// TIA Portal project "olbu" (V15)

(* hardware
DEVICE "S71500/ET200MP station_1"  S7-1500 station
   slot 0: "Rail_0"  Rack  6ES7 590-1***0-0AA0
   slot 1: "PLC_1"  CPU 1517F-3 PN/DP  6ES7 517-3FP00-0AB0  V2.5
      slot 3: "CPU display_1"  6ES7591-1BA00-0AA0
DEVICE "ET 200SP station_1"  ET 200SP-Station
   slot 0: "Rack_0"  Rack  6ES5 710-8MAx1
   slot 0: "volvo1606et200sp"  IM 155-6 PN ST  6ES7 155-6AU01-0BN0  V4.1
   slot 1: "DQ 8x24VDC/0.5A ST_1"  DQ 8x24VDC/0.5A ST  6ES7 132-6BF01-0BA0  V0.0
      slot 1: "DQ 8x24VDC/0.5A ST_1"  DQ 8x24VDC/0.5A ST
   slot 2: "DQ 8x24VDC/0.5A ST_2"  DQ 8x24VDC/0.5A ST  6ES7 132-6BF01-0BA0  V0.0
      slot 1: "DQ 8x24VDC/0.5A ST_2"  DQ 8x24VDC/0.5A ST
   slot 3: "DQ 8x24VDC/0.5A ST_3"  DQ 8x24VDC/0.5A ST  6ES7 132-6BF01-0BA0  V0.0
      slot 1: "DQ 8x24VDC/0.5A ST_3"  DQ 8x24VDC/0.5A ST
   slot 4: "Server module_1"  Server module  6ES7 193-6PA00-0AA0  V1.1
      slot 1: "Server module_1"  Server module
   slot 127: "BA 2xRJ45"  BA 2xRJ45  6ES7 193-6AR00-0AA0  V0.0
      slot 1: "Port_1"  6ES7 193-6AR00-0AA0  V0.0
      slot 2: "Port_2"  6ES7 193-6AR00-0AA0  V0.0
DEVICE "ET 200SP station_2"  ET 200SP-Station
   slot 0: "Rack_0"  Rack  6ES5 710-8MAx1
   slot 0: "volvo1607et200sp"  IM 155-6 PN ST  6ES7 155-6AU01-0BN0  V4.1
   slot 1: "DQ 8x24VDC/0.5A ST_1"  DQ 8x24VDC/0.5A ST  6ES7 132-6BF01-0BA0  V0.0
      slot 1: "DQ 8x24VDC/0.5A ST_1"  DQ 8x24VDC/0.5A ST
   slot 2: "DQ 8x24VDC/0.5A ST_2"  DQ 8x24VDC/0.5A ST  6ES7 132-6BF01-0BA0  V0.0
      slot 1: "DQ 8x24VDC/0.5A ST_2"  DQ 8x24VDC/0.5A ST
   slot 3: "DQ 8x24VDC/0.5A ST_3"  DQ 8x24VDC/0.5A ST  6ES7 132-6BF01-0BA0  V0.0
      slot 1: "DQ 8x24VDC/0.5A ST_3"  DQ 8x24VDC/0.5A ST
   slot 4: "Server module_1"  Server module  6ES7 193-6PA00-0AA0  V1.1
      slot 1: "Server module_1"  Server module
   slot 127: "BA 2xRJ45"  BA 2xRJ45  6ES7 193-6AR00-0AA0  V0.0
      slot 1: "Port_1"  6ES7 193-6AR00-0AA0  V0.0
      slot 2: "Port_2"  6ES7 193-6AR00-0AA0  V0.0
DEVICE "ET 200SP station_3"  ET 200SP-Station
   slot 0: "Rack_0"  Rack  6ES5 710-8MAx1
   slot 0: "volvo1608et200sp"  IM 155-6 PN ST  6ES7 155-6AU01-0BN0  V4.1
   slot 1: "DQ 8x24VDC/0.5A ST_1"  DQ 8x24VDC/0.5A ST  6ES7 132-6BF01-0BA0  V0.0
      slot 1: "DQ 8x24VDC/0.5A ST_1"  DQ 8x24VDC/0.5A ST
   slot 2: "DQ 8x24VDC/0.5A ST_2"  DQ 8x24VDC/0.5A ST  6ES7 132-6BF01-0BA0  V0.0
      slot 1: "DQ 8x24VDC/0.5A ST_2"  DQ 8x24VDC/0.5A ST
   slot 3: "DQ 8x24VDC/0.5A ST_3"  DQ 8x24VDC/0.5A ST  6ES7 132-6BF01-0BA0  V0.0
      slot 1: "DQ 8x24VDC/0.5A ST_3"  DQ 8x24VDC/0.5A ST
   slot 4: "Server module_1"  Server module  6ES7 193-6PA00-0AA0  V1.1
      slot 1: "Server module_1"  Server module
   slot 127: "BA 2xRJ45"  BA 2xRJ45  6ES7 193-6AR00-0AA0  V0.0
      slot 1: "Port_1"  6ES7 193-6AR00-0AA0  V0.0
      slot 2: "Port_2"  6ES7 193-6AR00-0AA0  V0.0
DEVICE "KP8_1"  SIMATIC Key Panel
   slot 0: "Rack"  Rail  V1.0
   slot 0: "volvo1608kp8"  KP8  6AV3 688-3AY36-0AX0  R01.00.00
DEVICE "KP8_2"  SIMATIC Key Panel
   slot 0: "Rack"  Rail  V1.0
   slot 0: "volvo1607kp8"  KP8  6AV3 688-3AY36-0AX0  R01.00.00
DEVICE "KP8_3"  SIMATIC Key Panel
   slot 0: "Rack"  Rail  V1.0
   slot 0: "volvo1606kp8"  KP8  6AV3 688-3AY36-0AX0  R01.00.00
DEVICE "KP8_4"  SIMATIC Key Panel
   slot 0: "Rack"  Rail  V1.0
   slot 0: "volvo1609kp8"  KP8  6AV3 688-3AY36-0AX0  R01.00.00
DEVICE "ET 200SP station_4"  ET 200SP-Station
   slot 0: "Rack_0"  Rack  6ES5 710-8MAx1
   slot 0: "volvo1609et200sp"  IM 155-6 PN ST  6ES7 155-6AU01-0BN0  V4.1
   slot 1: "DQ 8x24VDC/0.5A ST_1"  DQ 8x24VDC/0.5A ST  6ES7 132-6BF01-0BA0  V0.0
      slot 1: "DQ 8x24VDC/0.5A ST_1"  DQ 8x24VDC/0.5A ST
   slot 2: "DQ 8x24VDC/0.5A ST_2"  DQ 8x24VDC/0.5A ST  6ES7 132-6BF01-0BA0  V0.0
      slot 1: "DQ 8x24VDC/0.5A ST_2"  DQ 8x24VDC/0.5A ST
   slot 3: "DQ 8x24VDC/0.5A ST_3"  DQ 8x24VDC/0.5A ST  6ES7 132-6BF01-0BA0  V0.0
      slot 1: "DQ 8x24VDC/0.5A ST_3"  DQ 8x24VDC/0.5A ST
   slot 4: "Server module_1"  Server module  6ES7 193-6PA00-0AA0  V1.1
      slot 1: "Server module_1"  Server module
   slot 127: "BA 2xRJ45"  BA 2xRJ45  6ES7 193-6AR00-0AA0  V0.0
      slot 1: "Port_1"  6ES7 193-6AR00-0AA0  V0.0
      slot 2: "Port_2"  6ES7 193-6AR00-0AA0  V0.0
DEVICE "ET 200SP station_5"  ET 200SP-Station
   slot 0: "Rack_0"  Rack  6ES5 710-8MAx1
   slot 0: "volvo1610et200sp"  IM 155-6 PN ST  6ES7 155-6AU01-0BN0  V4.1
   slot 1: "DQ 8x24VDC/0.5A ST_1"  DQ 8x24VDC/0.5A ST  6ES7 132-6BF01-0BA0  V0.0
      slot 1: "DQ 8x24VDC/0.5A ST_1"  DQ 8x24VDC/0.5A ST
   slot 2: "DQ 8x24VDC/0.5A ST_2"  DQ 8x24VDC/0.5A ST  6ES7 132-6BF01-0BA0  V0.0
      slot 1: "DQ 8x24VDC/0.5A ST_2"  DQ 8x24VDC/0.5A ST
   slot 3: "DQ 8x24VDC/0.5A ST_3"  DQ 8x24VDC/0.5A ST  6ES7 132-6BF01-0BA0  V0.0
      slot 1: "DQ 8x24VDC/0.5A ST_3"  DQ 8x24VDC/0.5A ST
   slot 4: "Server module_1"  Server module  6ES7 193-6PA00-0AA0  V1.1
      slot 1: "Server module_1"  Server module
   slot 127: "BA 2xRJ45"  BA 2xRJ45  6ES7 193-6AR00-0AA0  V0.0
      slot 1: "Port_1"  6ES7 193-6AR00-0AA0  V0.0
      slot 2: "Port_2"  6ES7 193-6AR00-0AA0  V0.0
DEVICE "KP8_5"  SIMATIC Key Panel
   slot 0: "Rack"  Rail  V1.0
   slot 0: "volvo1610kp8"  KP8  6AV3 688-3AY36-0AX0  R01.00.00
DEVICE "ET 200SP station_6"  ET 200SP-Station
   slot 0: "Rack_0"  Rack  6ES5 710-8MAx1
   slot 0: "volvo1611et200sp"  IM 155-6 PN ST  6ES7 155-6AU01-0BN0  V4.1
   slot 1: "DQ 8x24VDC/0.5A ST_1"  DQ 8x24VDC/0.5A ST  6ES7 132-6BF01-0BA0  V0.0
      slot 1: "DQ 8x24VDC/0.5A ST_1"  DQ 8x24VDC/0.5A ST
   slot 2: "DQ 8x24VDC/0.5A ST_2"  DQ 8x24VDC/0.5A ST  6ES7 132-6BF01-0BA0  V0.0
      slot 1: "DQ 8x24VDC/0.5A ST_2"  DQ 8x24VDC/0.5A ST
   slot 3: "DQ 8x24VDC/0.5A ST_3"  DQ 8x24VDC/0.5A ST  6ES7 132-6BF01-0BA0  V0.0
      slot 1: "DQ 8x24VDC/0.5A ST_3"  DQ 8x24VDC/0.5A ST
   slot 4: "Server module_1"  Server module  6ES7 193-6PA00-0AA0  V1.1
      slot 1: "Server module_1"  Server module
   slot 127: "BA 2xRJ45"  BA 2xRJ45  6ES7 193-6AR00-0AA0  V0.0
      slot 1: "Port_1"  6ES7 193-6AR00-0AA0  V0.0
      slot 2: "Port_2"  6ES7 193-6AR00-0AA0  V0.0
DEVICE "KP8_6"  SIMATIC Key Panel
   slot 0: "Rack"  Rail  V1.0
   slot 0: "volvo1611kp8"  KP8  6AV3 688-3AY36-0AX0  R01.00.00
DEVICE "KP8_7"  SIMATIC Key Panel
   slot 0: "Rack"  Rail  V1.0
   slot 0: "volvo1601kp8"  KP8  6AV3 688-3AY36-0AX0  R01.00.00
DEVICE "ET 200SP station_7"  ET 200SP-Station
   slot 0: "Rack_0"  Rack  6ES5 710-8MAx1
   slot 0: "volvo1601et200sp"  IM 155-6 PN ST  6ES7 155-6AU01-0BN0  V4.1
   slot 1: "DQ 8x24VDC/0.5A ST_1"  DQ 8x24VDC/0.5A ST  6ES7 132-6BF01-0BA0  V0.0
      slot 1: "DQ 8x24VDC/0.5A ST_1"  DQ 8x24VDC/0.5A ST
   slot 2: "DQ 8x24VDC/0.5A ST_2"  DQ 8x24VDC/0.5A ST  6ES7 132-6BF01-0BA0  V0.0
      slot 1: "DQ 8x24VDC/0.5A ST_2"  DQ 8x24VDC/0.5A ST
   slot 3: "DQ 8x24VDC/0.5A ST_3"  DQ 8x24VDC/0.5A ST  6ES7 132-6BF01-0BA0  V0.0
      slot 1: "DQ 8x24VDC/0.5A ST_3"  DQ 8x24VDC/0.5A ST
   slot 4: "Server module_1"  Server module  6ES7 193-6PA00-0AA0  V1.1
      slot 1: "Server module_1"  Server module
   slot 127: "BA 2xRJ45"  BA 2xRJ45  6ES7 193-6AR00-0AA0  V0.0
      slot 1: "Port_1"  6ES7 193-6AR00-0AA0  V0.0
      slot 2: "Port_2"  6ES7 193-6AR00-0AA0  V0.0
DEVICE "KP8_8"  SIMATIC Key Panel
   slot 0: "Rack"  Rail  V1.0
   slot 0: "volvo1602kp8"  KP8  6AV3 688-3AY36-0AX0  R01.00.00
DEVICE "ET 200SP station_8"  ET 200SP-Station
   slot 0: "Rack_0"  Rack  6ES5 710-8MAx1
   slot 0: "volvo1602et200sp"  IM 155-6 PN ST  6ES7 155-6AU01-0BN0  V4.1
   slot 1: "DQ 8x24VDC/0.5A ST_1"  DQ 8x24VDC/0.5A ST  6ES7 132-6BF01-0BA0  V0.0
      slot 1: "DQ 8x24VDC/0.5A ST_1"  DQ 8x24VDC/0.5A ST
   slot 2: "DQ 8x24VDC/0.5A ST_2"  DQ 8x24VDC/0.5A ST  6ES7 132-6BF01-0BA0  V0.0
      slot 1: "DQ 8x24VDC/0.5A ST_2"  DQ 8x24VDC/0.5A ST
   slot 3: "DQ 8x24VDC/0.5A ST_3"  DQ 8x24VDC/0.5A ST  6ES7 132-6BF01-0BA0  V0.0
      slot 1: "DQ 8x24VDC/0.5A ST_3"  DQ 8x24VDC/0.5A ST
   slot 4: "Server module_1"  Server module  6ES7 193-6PA00-0AA0  V1.1
      slot 1: "Server module_1"  Server module
   slot 127: "BA 2xRJ45"  BA 2xRJ45  6ES7 193-6AR00-0AA0  V0.0
      slot 1: "Port_1"  6ES7 193-6AR00-0AA0  V0.0
      slot 2: "Port_2"  6ES7 193-6AR00-0AA0  V0.0
DEVICE "KP8_9"  SIMATIC Key Panel
   slot 0: "Rack"  Rail  V1.0
   slot 0: "volvo1603kp8"  KP8  6AV3 688-3AY36-0AX0  R01.00.00
DEVICE "ET 200SP station_9"  ET 200SP-Station
   slot 0: "Rack_0"  Rack  6ES5 710-8MAx1
   slot 0: "volvo1603et200sp"  IM 155-6 PN ST  6ES7 155-6AU01-0BN0  V4.1
   slot 1: "DQ 8x24VDC/0.5A ST_1"  DQ 8x24VDC/0.5A ST  6ES7 132-6BF01-0BA0  V0.0
      slot 1: "DQ 8x24VDC/0.5A ST_1"  DQ 8x24VDC/0.5A ST
   slot 2: "DQ 8x24VDC/0.5A ST_2"  DQ 8x24VDC/0.5A ST  6ES7 132-6BF01-0BA0  V0.0
      slot 1: "DQ 8x24VDC/0.5A ST_2"  DQ 8x24VDC/0.5A ST
   slot 3: "DQ 8x24VDC/0.5A ST_3"  DQ 8x24VDC/0.5A ST  6ES7 132-6BF01-0BA0  V0.0
      slot 1: "DQ 8x24VDC/0.5A ST_3"  DQ 8x24VDC/0.5A ST
   slot 4: "Server module_1"  Server module  6ES7 193-6PA00-0AA0  V1.1
      slot 1: "Server module_1"  Server module
   slot 127: "BA 2xRJ45"  BA 2xRJ45  6ES7 193-6AR00-0AA0  V0.0
      slot 1: "Port_1"  6ES7 193-6AR00-0AA0  V0.0
      slot 2: "Port_2"  6ES7 193-6AR00-0AA0  V0.0
DEVICE "KP8_10"  SIMATIC Key Panel
   slot 0: "Rack"  Rail  V1.0
   slot 0: "volvo1604kp8"  KP8  6AV3 688-3AY36-0AX0  R01.00.00
DEVICE "ET 200SP station_10"  ET 200SP-Station
   slot 0: "Rack_0"  Rack  6ES5 710-8MAx1
   slot 0: "volvo1604et200sp"  IM 155-6 PN ST  6ES7 155-6AU01-0BN0  V4.1
   slot 1: "DQ 8x24VDC/0.5A ST_1"  DQ 8x24VDC/0.5A ST  6ES7 132-6BF01-0BA0  V0.0
      slot 1: "DQ 8x24VDC/0.5A ST_1"  DQ 8x24VDC/0.5A ST
   slot 2: "DQ 8x24VDC/0.5A ST_2"  DQ 8x24VDC/0.5A ST  6ES7 132-6BF01-0BA0  V0.0
      slot 1: "DQ 8x24VDC/0.5A ST_2"  DQ 8x24VDC/0.5A ST
   slot 3: "DQ 8x24VDC/0.5A ST_3"  DQ 8x24VDC/0.5A ST  6ES7 132-6BF01-0BA0  V0.0
      slot 1: "DQ 8x24VDC/0.5A ST_3"  DQ 8x24VDC/0.5A ST
   slot 4: "Server module_1"  Server module  6ES7 193-6PA00-0AA0  V1.1
      slot 1: "Server module_1"  Server module
   slot 127: "BA 2xRJ45"  BA 2xRJ45  6ES7 193-6AR00-0AA0  V0.0
      slot 1: "Port_1"  6ES7 193-6AR00-0AA0  V0.0
      slot 2: "Port_2"  6ES7 193-6AR00-0AA0  V0.0
DEVICE "KP8_11"  SIMATIC Key Panel
   slot 0: "Rack"  Rail  V1.0
   slot 0: "volvo1605kp8"  KP8  6AV3 688-3AY36-0AX0  R01.00.00
DEVICE "ET 200SP station_11"  ET 200SP-Station
   slot 0: "Rack_0"  Rack  6ES5 710-8MAx1
   slot 0: "volvo1605et200sp"  IM 155-6 PN ST  6ES7 155-6AU01-0BN0  V4.1
   slot 1: "DQ 8x24VDC/0.5A ST_1"  DQ 8x24VDC/0.5A ST  6ES7 132-6BF01-0BA0  V0.0
      slot 1: "DQ 8x24VDC/0.5A ST_1"  DQ 8x24VDC/0.5A ST
   slot 2: "DQ 8x24VDC/0.5A ST_2"  DQ 8x24VDC/0.5A ST  6ES7 132-6BF01-0BA0  V0.0
      slot 1: "DQ 8x24VDC/0.5A ST_2"  DQ 8x24VDC/0.5A ST
   slot 3: "DQ 8x24VDC/0.5A ST_3"  DQ 8x24VDC/0.5A ST  6ES7 132-6BF01-0BA0  V0.0
      slot 1: "DQ 8x24VDC/0.5A ST_3"  DQ 8x24VDC/0.5A ST
   slot 4: "Server module_1"  Server module  6ES7 193-6PA00-0AA0  V1.1
      slot 1: "Server module_1"  Server module
   slot 127: "BA 2xRJ45"  BA 2xRJ45  6ES7 193-6AR00-0AA0  V0.0
      slot 1: "Port_1"  6ES7 193-6AR00-0AA0  V0.0
      slot 2: "Port_2"  6ES7 193-6AR00-0AA0  V0.0
DEVICE "KP8_12"  SIMATIC Key Panel
   slot 0: "Rack"  Rail  V1.0
   slot 0: "chm02kp8"  KP8  6AV3 688-3AY36-0AX0  R01.00.00
DEVICE "ET 200SP station_12"  ET 200SP-Station
   slot 0: "Rack_0"  Rack  6ES5 710-8MAx1
   slot 0: "chm02et200sp"  IM 155-6 PN ST  6ES7 155-6AU01-0BN0  V4.1
   slot 1: "DQ 8x24VDC/0.5A ST_1"  DQ 8x24VDC/0.5A ST  6ES7 132-6BF01-0BA0  V0.0
      slot 1: "DQ 8x24VDC/0.5A ST_1"  DQ 8x24VDC/0.5A ST
   slot 2: "DQ 8x24VDC/0.5A ST_2"  DQ 8x24VDC/0.5A ST  6ES7 132-6BF01-0BA0  V0.0
      slot 1: "DQ 8x24VDC/0.5A ST_2"  DQ 8x24VDC/0.5A ST
   slot 3: "DQ 8x24VDC/0.5A ST_3"  DQ 8x24VDC/0.5A ST  6ES7 132-6BF01-0BA0  V0.0
      slot 1: "DQ 8x24VDC/0.5A ST_3"  DQ 8x24VDC/0.5A ST
   slot 4: "Server module_1"  Server module  6ES7 193-6PA00-0AA0  V1.1
      slot 1: "Server module_1"  Server module
   slot 127: "BA 2xRJ45"  BA 2xRJ45  6ES7 193-6AR00-0AA0  V0.0
      slot 1: "Port_1"  6ES7 193-6AR00-0AA0  V0.0
      slot 2: "Port_2"  6ES7 193-6AR00-0AA0  V0.0
DEVICE "KP8_13"  SIMATIC Key Panel
   slot 0: "Rack"  Rail  V1.0
   slot 0: "chm03kp8"  KP8  6AV3 688-3AY36-0AX0  R01.00.00
DEVICE "ET 200SP station_13"  ET 200SP-Station
   slot 0: "Rack_0"  Rack  6ES5 710-8MAx1
   slot 0: "chm03et200sp"  IM 155-6 PN ST  6ES7 155-6AU01-0BN0  V4.1
   slot 1: "DQ 8x24VDC/0.5A ST_1"  DQ 8x24VDC/0.5A ST  6ES7 132-6BF01-0BA0  V0.0
      slot 1: "DQ 8x24VDC/0.5A ST_1"  DQ 8x24VDC/0.5A ST
   slot 2: "DQ 8x24VDC/0.5A ST_2"  DQ 8x24VDC/0.5A ST  6ES7 132-6BF01-0BA0  V0.0
      slot 1: "DQ 8x24VDC/0.5A ST_2"  DQ 8x24VDC/0.5A ST
   slot 3: "DQ 8x24VDC/0.5A ST_3"  DQ 8x24VDC/0.5A ST  6ES7 132-6BF01-0BA0  V0.0
      slot 1: "DQ 8x24VDC/0.5A ST_3"  DQ 8x24VDC/0.5A ST
   slot 4: "Server module_1"  Server module  6ES7 193-6PA00-0AA0  V1.1
      slot 1: "Server module_1"  Server module
   slot 127: "BA 2xRJ45"  BA 2xRJ45  6ES7 193-6AR00-0AA0  V0.0
      slot 1: "Port_1"  6ES7 193-6AR00-0AA0  V0.0
      slot 2: "Port_2"  6ES7 193-6AR00-0AA0  V0.0
DEVICE "KP8_14"  SIMATIC Key Panel
   slot 0: "Rack"  Rail  V1.0
   slot 0: "chm04kp8"  KP8  6AV3 688-3AY36-0AX0  R01.00.00
DEVICE "ET 200SP station_14"  ET 200SP-Station
   slot 0: "Rack_0"  Rack  6ES5 710-8MAx1
   slot 0: "chm04et200sp"  IM 155-6 PN ST  6ES7 155-6AU01-0BN0  V4.1
   slot 1: "DQ 8x24VDC/0.5A ST_1"  DQ 8x24VDC/0.5A ST  6ES7 132-6BF01-0BA0  V0.0
      slot 1: "DQ 8x24VDC/0.5A ST_1"  DQ 8x24VDC/0.5A ST
   slot 2: "DQ 8x24VDC/0.5A ST_2"  DQ 8x24VDC/0.5A ST  6ES7 132-6BF01-0BA0  V0.0
      slot 1: "DQ 8x24VDC/0.5A ST_2"  DQ 8x24VDC/0.5A ST
   slot 3: "DQ 8x24VDC/0.5A ST_3"  DQ 8x24VDC/0.5A ST  6ES7 132-6BF01-0BA0  V0.0
      slot 1: "DQ 8x24VDC/0.5A ST_3"  DQ 8x24VDC/0.5A ST
   slot 4: "Server module_1"  Server module  6ES7 193-6PA00-0AA0  V1.1
      slot 1: "Server module_1"  Server module
   slot 127: "BA 2xRJ45"  BA 2xRJ45  6ES7 193-6AR00-0AA0  V0.0
      slot 1: "Port_1"  6ES7 193-6AR00-0AA0  V0.0
      slot 2: "Port_2"  6ES7 193-6AR00-0AA0  V0.0
DEVICE "KP8_15"  SIMATIC Key Panel
   slot 0: "Rack"  Rail  V1.0
   slot 0: "chm05kp8"  KP8  6AV3 688-3AY36-0AX0  R01.00.00
DEVICE "ET 200SP station_15"  ET 200SP-Station
   slot 0: "Rack_0"  Rack  6ES5 710-8MAx1
   slot 0: "chm05et200sp"  IM 155-6 PN ST  6ES7 155-6AU01-0BN0  V4.1
   slot 1: "DQ 8x24VDC/0.5A ST_1"  DQ 8x24VDC/0.5A ST  6ES7 132-6BF01-0BA0  V0.0
      slot 1: "DQ 8x24VDC/0.5A ST_1"  DQ 8x24VDC/0.5A ST
   slot 2: "DQ 8x24VDC/0.5A ST_2"  DQ 8x24VDC/0.5A ST  6ES7 132-6BF01-0BA0  V0.0
      slot 1: "DQ 8x24VDC/0.5A ST_2"  DQ 8x24VDC/0.5A ST
   slot 3: "DQ 8x24VDC/0.5A ST_3"  DQ 8x24VDC/0.5A ST  6ES7 132-6BF01-0BA0  V0.0
      slot 1: "DQ 8x24VDC/0.5A ST_3"  DQ 8x24VDC/0.5A ST
   slot 4: "Server module_1"  Server module  6ES7 193-6PA00-0AA0  V1.1
      slot 1: "Server module_1"  Server module
   slot 127: "BA 2xRJ45"  BA 2xRJ45  6ES7 193-6AR00-0AA0  V0.0
      slot 1: "Port_1"  6ES7 193-6AR00-0AA0  V0.0
      slot 2: "Port_2"  6ES7 193-6AR00-0AA0  V0.0
DEVICE "KP8_16"  SIMATIC Key Panel
   slot 0: "Rack"  Rail  V1.0
   slot 0: "cdo01kp8"  KP8  6AV3 688-3AY36-0AX0  R01.00.00
DEVICE "ET 200SP station_16"  ET 200SP-Station
   slot 0: "Rack_0"  Rack  6ES5 710-8MAx1
   slot 0: "cdo01et200sp"  IM 155-6 PN ST  6ES7 155-6AU01-0BN0  V4.1
   slot 1: "DQ 8x24VDC/0.5A ST_1"  DQ 8x24VDC/0.5A ST  6ES7 132-6BF01-0BA0  V0.0
      slot 1: "DQ 8x24VDC/0.5A ST_1"  DQ 8x24VDC/0.5A ST
   slot 2: "DQ 8x24VDC/0.5A ST_2"  DQ 8x24VDC/0.5A ST  6ES7 132-6BF01-0BA0  V0.0
      slot 1: "DQ 8x24VDC/0.5A ST_2"  DQ 8x24VDC/0.5A ST
   slot 3: "DQ 8x24VDC/0.5A ST_3"  DQ 8x24VDC/0.5A ST  6ES7 132-6BF01-0BA0  V0.0
      slot 1: "DQ 8x24VDC/0.5A ST_3"  DQ 8x24VDC/0.5A ST
   slot 4: "Server module_1"  Server module  6ES7 193-6PA00-0AA0  V1.1
      slot 1: "Server module_1"  Server module
   slot 127: "BA 2xRJ45"  BA 2xRJ45  6ES7 193-6AR00-0AA0  V0.0
      slot 1: "Port_1"  6ES7 193-6AR00-0AA0  V0.0
      slot 2: "Port_2"  6ES7 193-6AR00-0AA0  V0.0
DEVICE "KP8_17"  SIMATIC Key Panel
   slot 0: "Rack"  Rail  V1.0
   slot 0: "cdo02kp8"  KP8  6AV3 688-3AY36-0AX0  R01.00.00
DEVICE "ET 200SP station_17"  ET 200SP-Station
   slot 0: "Rack_0"  Rack  6ES5 710-8MAx1
   slot 0: "cdo02et200sp"  IM 155-6 PN ST  6ES7 155-6AU01-0BN0  V4.1
   slot 1: "DQ 8x24VDC/0.5A ST_1"  DQ 8x24VDC/0.5A ST  6ES7 132-6BF01-0BA0  V0.0
      slot 1: "DQ 8x24VDC/0.5A ST_1"  DQ 8x24VDC/0.5A ST
   slot 2: "DQ 8x24VDC/0.5A ST_2"  DQ 8x24VDC/0.5A ST  6ES7 132-6BF01-0BA0  V0.0
      slot 1: "DQ 8x24VDC/0.5A ST_2"  DQ 8x24VDC/0.5A ST
   slot 3: "DQ 8x24VDC/0.5A ST_3"  DQ 8x24VDC/0.5A ST  6ES7 132-6BF01-0BA0  V0.0
      slot 1: "DQ 8x24VDC/0.5A ST_3"  DQ 8x24VDC/0.5A ST
   slot 4: "Server module_1"  Server module  6ES7 193-6PA00-0AA0  V1.1
      slot 1: "Server module_1"  Server module
   slot 127: "BA 2xRJ45"  BA 2xRJ45  6ES7 193-6AR00-0AA0  V0.0
      slot 1: "Port_1"  6ES7 193-6AR00-0AA0  V0.0
      slot 2: "Port_2"  6ES7 193-6AR00-0AA0  V0.0
DEVICE "KP8_18"  SIMATIC Key Panel
   slot 0: "Rack"  Rail  V1.0
   slot 0: "cdo03kp8"  KP8  6AV3 688-3AY36-0AX0  R01.00.00
DEVICE "ET 200SP station_18"  ET 200SP-Station
   slot 0: "Rack_0"  Rack  6ES5 710-8MAx1
   slot 0: "cdo03et200sp"  IM 155-6 PN ST  6ES7 155-6AU01-0BN0  V4.1
   slot 1: "DQ 8x24VDC/0.5A ST_1"  DQ 8x24VDC/0.5A ST  6ES7 132-6BF01-0BA0  V0.0
      slot 1: "DQ 8x24VDC/0.5A ST_1"  DQ 8x24VDC/0.5A ST
   slot 2: "DQ 8x24VDC/0.5A ST_2"  DQ 8x24VDC/0.5A ST  6ES7 132-6BF01-0BA0  V0.0
      slot 1: "DQ 8x24VDC/0.5A ST_2"  DQ 8x24VDC/0.5A ST
   slot 3: "DQ 8x24VDC/0.5A ST_3"  DQ 8x24VDC/0.5A ST  6ES7 132-6BF01-0BA0  V0.0
      slot 1: "DQ 8x24VDC/0.5A ST_3"  DQ 8x24VDC/0.5A ST
   slot 4: "Server module_1"  Server module  6ES7 193-6PA00-0AA0  V1.1
      slot 1: "Server module_1"  Server module
   slot 127: "BA 2xRJ45"  BA 2xRJ45  6ES7 193-6AR00-0AA0  V0.0
      slot 1: "Port_1"  6ES7 193-6AR00-0AA0  V0.0
      slot 2: "Port_2"  6ES7 193-6AR00-0AA0  V0.0
DEVICE "KP8_19"  SIMATIC Key Panel
   slot 0: "Rack"  Rail  V1.0
   slot 0: "bfl01kp8"  KP8  6AV3 688-3AY36-0AX0  R01.00.00
DEVICE "ET 200SP station_19"  ET 200SP-Station
   slot 0: "Rack_0"  Rack  6ES5 710-8MAx1
   slot 0: "bfl01et200sp"  IM 155-6 PN ST  6ES7 155-6AU01-0BN0  V4.1
   slot 1: "DQ 8x24VDC/0.5A ST_1"  DQ 8x24VDC/0.5A ST  6ES7 132-6BF01-0BA0  V0.0
      slot 1: "DQ 8x24VDC/0.5A ST_1"  DQ 8x24VDC/0.5A ST
   slot 2: "DQ 8x24VDC/0.5A ST_2"  DQ 8x24VDC/0.5A ST  6ES7 132-6BF01-0BA0  V0.0
      slot 1: "DQ 8x24VDC/0.5A ST_2"  DQ 8x24VDC/0.5A ST
   slot 3: "DQ 8x24VDC/0.5A ST_3"  DQ 8x24VDC/0.5A ST  6ES7 132-6BF01-0BA0  V0.0
      slot 1: "DQ 8x24VDC/0.5A ST_3"  DQ 8x24VDC/0.5A ST
   slot 4: "Server module_1"  Server module  6ES7 193-6PA00-0AA0  V1.1
      slot 1: "Server module_1"  Server module
   slot 127: "BA 2xRJ45"  BA 2xRJ45  6ES7 193-6AR00-0AA0  V0.0
      slot 1: "Port_1"  6ES7 193-6AR00-0AA0  V0.0
      slot 2: "Port_2"  6ES7 193-6AR00-0AA0  V0.0
DEVICE "KP8_20"  SIMATIC Key Panel
   slot 0: "Rack"  Rail  V1.0
   slot 0: "bfl02kp8"  KP8  6AV3 688-3AY36-0AX0  R01.00.00
DEVICE "ET 200SP station_20"  ET 200SP-Station
   slot 0: "Rack_0"  Rack  6ES5 710-8MAx1
   slot 0: "bfl02et200sp"  IM 155-6 PN ST  6ES7 155-6AU01-0BN0  V4.1
   slot 1: "DQ 8x24VDC/0.5A ST_1"  DQ 8x24VDC/0.5A ST  6ES7 132-6BF01-0BA0  V0.0
      slot 1: "DQ 8x24VDC/0.5A ST_1"  DQ 8x24VDC/0.5A ST
   slot 2: "DQ 8x24VDC/0.5A ST_2"  DQ 8x24VDC/0.5A ST  6ES7 132-6BF01-0BA0  V0.0
      slot 1: "DQ 8x24VDC/0.5A ST_2"  DQ 8x24VDC/0.5A ST
   slot 3: "DQ 8x24VDC/0.5A ST_3"  DQ 8x24VDC/0.5A ST  6ES7 132-6BF01-0BA0  V0.0
      slot 1: "DQ 8x24VDC/0.5A ST_3"  DQ 8x24VDC/0.5A ST
   slot 4: "Server module_1"  Server module  6ES7 193-6PA00-0AA0  V1.1
      slot 1: "Server module_1"  Server module
   slot 127: "BA 2xRJ45"  BA 2xRJ45  6ES7 193-6AR00-0AA0  V0.0
      slot 1: "Port_1"  6ES7 193-6AR00-0AA0  V0.0
      slot 2: "Port_2"  6ES7 193-6AR00-0AA0  V0.0
DEVICE "KP8_21"  SIMATIC Key Panel
   slot 0: "Rack"  Rail  V1.0
   slot 0: "bfl03kp8"  KP8  6AV3 688-3AY36-0AX0  R01.00.00
DEVICE "ET 200SP station_21"  ET 200SP-Station
   slot 0: "Rack_0"  Rack  6ES5 710-8MAx1
   slot 0: "bfl03et200sp"  IM 155-6 PN ST  6ES7 155-6AU01-0BN0  V4.1
   slot 1: "DQ 8x24VDC/0.5A ST_1"  DQ 8x24VDC/0.5A ST  6ES7 132-6BF01-0BA0  V0.0
      slot 1: "DQ 8x24VDC/0.5A ST_1"  DQ 8x24VDC/0.5A ST
   slot 2: "DQ 8x24VDC/0.5A ST_2"  DQ 8x24VDC/0.5A ST  6ES7 132-6BF01-0BA0  V0.0
      slot 1: "DQ 8x24VDC/0.5A ST_2"  DQ 8x24VDC/0.5A ST
   slot 3: "DQ 8x24VDC/0.5A ST_3"  DQ 8x24VDC/0.5A ST  6ES7 132-6BF01-0BA0  V0.0
      slot 1: "DQ 8x24VDC/0.5A ST_3"  DQ 8x24VDC/0.5A ST
   slot 4: "Server module_1"  Server module  6ES7 193-6PA00-0AA0  V1.1
      slot 1: "Server module_1"  Server module
   slot 127: "BA 2xRJ45"  BA 2xRJ45  6ES7 193-6AR00-0AA0  V0.0
      slot 1: "Port_1"  6ES7 193-6AR00-0AA0  V0.0
      slot 2: "Port_2"  6ES7 193-6AR00-0AA0  V0.0
DEVICE "KP8_22"  SIMATIC Key Panel
   slot 0: "Rack"  Rail  V1.0
   slot 0: "lgs01kp8"  KP8  6AV3 688-3AY36-0AX0  R01.00.00
DEVICE "ET 200SP station_22"  ET 200SP-Station
   slot 0: "Rack_0"  Rack  6ES5 710-8MAx1
   slot 0: "lgs01et200sp"  IM 155-6 PN ST  6ES7 155-6AU01-0BN0  V4.1
   slot 1: "DQ 8x24VDC/0.5A ST_1"  DQ 8x24VDC/0.5A ST  6ES7 132-6BF01-0BA0  V0.0
      slot 1: "DQ 8x24VDC/0.5A ST_1"  DQ 8x24VDC/0.5A ST
   slot 2: "DQ 8x24VDC/0.5A ST_2"  DQ 8x24VDC/0.5A ST  6ES7 132-6BF01-0BA0  V0.0
      slot 1: "DQ 8x24VDC/0.5A ST_2"  DQ 8x24VDC/0.5A ST
   slot 3: "DQ 8x24VDC/0.5A ST_3"  DQ 8x24VDC/0.5A ST  6ES7 132-6BF01-0BA0  V0.0
      slot 1: "DQ 8x24VDC/0.5A ST_3"  DQ 8x24VDC/0.5A ST
   slot 4: "Server module_1"  Server module  6ES7 193-6PA00-0AA0  V1.1
      slot 1: "Server module_1"  Server module
   slot 127: "BA 2xRJ45"  BA 2xRJ45  6ES7 193-6AR00-0AA0  V0.0
      slot 1: "Port_1"  6ES7 193-6AR00-0AA0  V0.0
      slot 2: "Port_2"  6ES7 193-6AR00-0AA0  V0.0
DEVICE "KP8_23"  SIMATIC Key Panel
   slot 0: "Rack"  Rail  V1.0
   slot 0: "lgs02kp8"  KP8  6AV3 688-3AY36-0AX0  R01.00.00
DEVICE "ET 200SP station_23"  ET 200SP-Station
   slot 0: "Rack_0"  Rack  6ES5 710-8MAx1
   slot 0: "lgs02et200sp"  IM 155-6 PN ST  6ES7 155-6AU01-0BN0  V4.1
   slot 1: "DQ 8x24VDC/0.5A ST_1"  DQ 8x24VDC/0.5A ST  6ES7 132-6BF01-0BA0  V0.0
      slot 1: "DQ 8x24VDC/0.5A ST_1"  DQ 8x24VDC/0.5A ST
   slot 2: "DQ 8x24VDC/0.5A ST_2"  DQ 8x24VDC/0.5A ST  6ES7 132-6BF01-0BA0  V0.0
      slot 1: "DQ 8x24VDC/0.5A ST_2"  DQ 8x24VDC/0.5A ST
   slot 3: "DQ 8x24VDC/0.5A ST_3"  DQ 8x24VDC/0.5A ST  6ES7 132-6BF01-0BA0  V0.0
      slot 1: "DQ 8x24VDC/0.5A ST_3"  DQ 8x24VDC/0.5A ST
   slot 4: "Server module_1"  Server module  6ES7 193-6PA00-0AA0  V1.1
      slot 1: "Server module_1"  Server module
   slot 127: "BA 2xRJ45"  BA 2xRJ45  6ES7 193-6AR00-0AA0  V0.0
      slot 1: "Port_1"  6ES7 193-6AR00-0AA0  V0.0
      slot 2: "Port_2"  6ES7 193-6AR00-0AA0  V0.0
DEVICE "KP8_24"  SIMATIC Key Panel
   slot 0: "Rack"  Rail  V1.0
   slot 0: "chm01kp8"  KP8  6AV3 688-3AY36-0AX0  R01.00.00
DEVICE "ET 200SP station_24"  ET 200SP-Station
   slot 0: "Rack_0"  Rack  6ES5 710-8MAx1
   slot 0: "chm01et200sp"  IM 155-6 PN ST  6ES7 155-6AU01-0BN0  V4.1
   slot 1: "DQ 8x24VDC/0.5A ST_1"  DQ 8x24VDC/0.5A ST  6ES7 132-6BF01-0BA0  V0.0
      slot 1: "DQ 8x24VDC/0.5A ST_1"  DQ 8x24VDC/0.5A ST
   slot 2: "DQ 8x24VDC/0.5A ST_2"  DQ 8x24VDC/0.5A ST  6ES7 132-6BF01-0BA0  V0.0
      slot 1: "DQ 8x24VDC/0.5A ST_2"  DQ 8x24VDC/0.5A ST
   slot 3: "DQ 8x24VDC/0.5A ST_3"  DQ 8x24VDC/0.5A ST  6ES7 132-6BF01-0BA0  V0.0
      slot 1: "DQ 8x24VDC/0.5A ST_3"  DQ 8x24VDC/0.5A ST
   slot 4: "Server module_1"  Server module  6ES7 193-6PA00-0AA0  V1.1
      slot 1: "Server module_1"  Server module
   slot 127: "BA 2xRJ45"  BA 2xRJ45  6ES7 193-6AR00-0AA0  V0.0
      slot 1: "Port_1"  6ES7 193-6AR00-0AA0  V0.0
      slot 2: "Port_2"  6ES7 193-6AR00-0AA0  V0.0
DEVICE "KP8_25"  SIMATIC Key Panel
   slot 0: "Rack"  Rail  V1.0
   slot 0: "lgs03kp8"  KP8  6AV3 688-3AY36-0AX0  R01.00.00
DEVICE "ET 200SP station_25"  ET 200SP-Station
   slot 0: "Rack_0"  Rack  6ES5 710-8MAx1
   slot 0: "lgs03et200sp"  IM 155-6 PN ST  6ES7 155-6AU01-0BN0  V4.1
   slot 1: "DQ 8x24VDC/0.5A ST_1"  DQ 8x24VDC/0.5A ST  6ES7 132-6BF01-0BA0  V0.0
      slot 1: "DQ 8x24VDC/0.5A ST_1"  DQ 8x24VDC/0.5A ST
   slot 2: "DQ 8x24VDC/0.5A ST_2"  DQ 8x24VDC/0.5A ST  6ES7 132-6BF01-0BA0  V0.0
      slot 1: "DQ 8x24VDC/0.5A ST_2"  DQ 8x24VDC/0.5A ST
   slot 3: "DQ 8x24VDC/0.5A ST_3"  DQ 8x24VDC/0.5A ST  6ES7 132-6BF01-0BA0  V0.0
      slot 1: "DQ 8x24VDC/0.5A ST_3"  DQ 8x24VDC/0.5A ST
   slot 4: "Server module_1"  Server module  6ES7 193-6PA00-0AA0  V1.1
      slot 1: "Server module_1"  Server module
   slot 127: "BA 2xRJ45"  BA 2xRJ45  6ES7 193-6AR00-0AA0  V0.0
      slot 1: "Port_1"  6ES7 193-6AR00-0AA0  V0.0
      slot 2: "Port_2"  6ES7 193-6AR00-0AA0  V0.0
DEVICE "KP8_26"  SIMATIC Key Panel
   slot 0: "Rack"  Rail  V1.0
   slot 0: "pc02kp8"  KP8  6AV3 688-3AY36-0AX0  R01.00.00
DEVICE "ET 200SP station_26"  ET 200SP-Station
   slot 0: "Rack_0"  Rack  6ES5 710-8MAx1
   slot 0: "cv01et200sp"  IM 155-6 PN ST  6ES7 155-6AU01-0BN0  V4.1
   slot 1: "DQ 8x24VDC/0.5A ST_1"  DQ 8x24VDC/0.5A ST  6ES7 132-6BF01-0BA0  V0.0
      slot 1: "DQ 8x24VDC/0.5A ST_1"  DQ 8x24VDC/0.5A ST
   slot 2: "DQ 8x24VDC/0.5A ST_2"  DQ 8x24VDC/0.5A ST  6ES7 132-6BF01-0BA0  V0.0
      slot 1: "DQ 8x24VDC/0.5A ST_2"  DQ 8x24VDC/0.5A ST
   slot 3: "DQ 8x24VDC/0.5A ST_3"  DQ 8x24VDC/0.5A ST  6ES7 132-6BF01-0BA0  V0.0
      slot 1: "DQ 8x24VDC/0.5A ST_3"  DQ 8x24VDC/0.5A ST
   slot 4: "Server module_1"  Server module  6ES7 193-6PA00-0AA0  V1.1
      slot 1: "Server module_1"  Server module
   slot 127: "BA 2xRJ45"  BA 2xRJ45  6ES7 193-6AR00-0AA0  V0.0
      slot 1: "Port_1"  6ES7 193-6AR00-0AA0  V0.0
      slot 2: "Port_2"  6ES7 193-6AR00-0AA0  V0.0
DEVICE "ET 200SP station_27"  ET 200SP-Station
   slot 0: "Rack_0"  Rack  6ES5 710-8MAx1
   slot 0: "cv02et200sp"  IM 155-6 PN ST  6ES7 155-6AU01-0BN0  V4.1
   slot 1: "DQ 8x24VDC/0.5A ST_1"  DQ 8x24VDC/0.5A ST  6ES7 132-6BF01-0BA0  V0.0
      slot 1: "DQ 8x24VDC/0.5A ST_1"  DQ 8x24VDC/0.5A ST
   slot 2: "DQ 8x24VDC/0.5A ST_2"  DQ 8x24VDC/0.5A ST  6ES7 132-6BF01-0BA0  V0.0
      slot 1: "DQ 8x24VDC/0.5A ST_2"  DQ 8x24VDC/0.5A ST
   slot 3: "DQ 8x24VDC/0.5A ST_3"  DQ 8x24VDC/0.5A ST  6ES7 132-6BF01-0BA0  V0.0
      slot 1: "DQ 8x24VDC/0.5A ST_3"  DQ 8x24VDC/0.5A ST
   slot 4: "Server module_1"  Server module  6ES7 193-6PA00-0AA0  V1.1
      slot 1: "Server module_1"  Server module
   slot 127: "BA 2xRJ45"  BA 2xRJ45  6ES7 193-6AR00-0AA0  V0.0
      slot 1: "Port_1"  6ES7 193-6AR00-0AA0  V0.0
      slot 2: "Port_2"  6ES7 193-6AR00-0AA0  V0.0
DEVICE "ET 200SP station_28"  ET 200SP-Station
   slot 0: "Rack_0"  Rack  6ES5 710-8MAx1
   slot 0: "cv03et200sp"  IM 155-6 PN ST  6ES7 155-6AU01-0BN0  V4.1
   slot 1: "DQ 8x24VDC/0.5A ST_1"  DQ 8x24VDC/0.5A ST  6ES7 132-6BF01-0BA0  V0.0
      slot 1: "DQ 8x24VDC/0.5A ST_1"  DQ 8x24VDC/0.5A ST
   slot 2: "DQ 8x24VDC/0.5A ST_2"  DQ 8x24VDC/0.5A ST  6ES7 132-6BF01-0BA0  V0.0
      slot 1: "DQ 8x24VDC/0.5A ST_2"  DQ 8x24VDC/0.5A ST
   slot 3: "DQ 8x24VDC/0.5A ST_3"  DQ 8x24VDC/0.5A ST  6ES7 132-6BF01-0BA0  V0.0
      slot 1: "DQ 8x24VDC/0.5A ST_3"  DQ 8x24VDC/0.5A ST
   slot 4: "Server module_1"  Server module  6ES7 193-6PA00-0AA0  V1.1
      slot 1: "Server module_1"  Server module
   slot 127: "BA 2xRJ45"  BA 2xRJ45  6ES7 193-6AR00-0AA0  V0.0
      slot 1: "Port_1"  6ES7 193-6AR00-0AA0  V0.0
      slot 2: "Port_2"  6ES7 193-6AR00-0AA0  V0.0
DEVICE "ET 200SP station_29"  ET 200SP-Station
   slot 0: "Rack_0"  Rack  6ES5 710-8MAx1
   slot 0: "cv04et200sp"  IM 155-6 PN ST  6ES7 155-6AU01-0BN0  V4.1
   slot 1: "DQ 8x24VDC/0.5A ST_1"  DQ 8x24VDC/0.5A ST  6ES7 132-6BF01-0BA0  V0.0
      slot 1: "DQ 8x24VDC/0.5A ST_1"  DQ 8x24VDC/0.5A ST
   slot 2: "DQ 8x24VDC/0.5A ST_2"  DQ 8x24VDC/0.5A ST  6ES7 132-6BF01-0BA0  V0.0
      slot 1: "DQ 8x24VDC/0.5A ST_2"  DQ 8x24VDC/0.5A ST
   slot 3: "DQ 8x24VDC/0.5A ST_3"  DQ 8x24VDC/0.5A ST  6ES7 132-6BF01-0BA0  V0.0
      slot 1: "DQ 8x24VDC/0.5A ST_3"  DQ 8x24VDC/0.5A ST
   slot 4: "Server module_1"  Server module  6ES7 193-6PA00-0AA0  V1.1
      slot 1: "Server module_1"  Server module
   slot 127: "BA 2xRJ45"  BA 2xRJ45  6ES7 193-6AR00-0AA0  V0.0
      slot 1: "Port_1"  6ES7 193-6AR00-0AA0  V0.0
      slot 2: "Port_2"  6ES7 193-6AR00-0AA0  V0.0
DEVICE "ET 200SP station_30"  ET 200SP-Station
   slot 0: "Rack_0"  Rack  6ES5 710-8MAx1
   slot 0: "pc01et200sp"  IM 155-6 PN ST  6ES7 155-6AU01-0BN0  V4.1
   slot 1: "DQ 8x24VDC/0.5A ST_1"  DQ 8x24VDC/0.5A ST  6ES7 132-6BF01-0BA0  V0.0
      slot 1: "DQ 8x24VDC/0.5A ST_1"  DQ 8x24VDC/0.5A ST
   slot 2: "DQ 8x24VDC/0.5A ST_2"  DQ 8x24VDC/0.5A ST  6ES7 132-6BF01-0BA0  V0.0
      slot 1: "DQ 8x24VDC/0.5A ST_2"  DQ 8x24VDC/0.5A ST
   slot 3: "DQ 8x24VDC/0.5A ST_3"  DQ 8x24VDC/0.5A ST  6ES7 132-6BF01-0BA0  V0.0
      slot 1: "DQ 8x24VDC/0.5A ST_3"  DQ 8x24VDC/0.5A ST
   slot 4: "Server module_1"  Server module  6ES7 193-6PA00-0AA0  V1.1
      slot 1: "Server module_1"  Server module
   slot 127: "BA 2xRJ45"  BA 2xRJ45  6ES7 193-6AR00-0AA0  V0.0
      slot 1: "Port_1"  6ES7 193-6AR00-0AA0  V0.0
      slot 2: "Port_2"  6ES7 193-6AR00-0AA0  V0.0
DEVICE "ET 200SP station_31"  ET 200SP-Station
   slot 0: "Rack_0"  Rack  6ES5 710-8MAx1
   slot 0: "pc02et200sp"  IM 155-6 PN ST  6ES7 155-6AU01-0BN0  V4.1
   slot 1: "DQ 8x24VDC/0.5A ST_1"  DQ 8x24VDC/0.5A ST  6ES7 132-6BF01-0BA0  V0.0
      slot 1: "DQ 8x24VDC/0.5A ST_1"  DQ 8x24VDC/0.5A ST
   slot 2: "DQ 8x24VDC/0.5A ST_2"  DQ 8x24VDC/0.5A ST  6ES7 132-6BF01-0BA0  V0.0
      slot 1: "DQ 8x24VDC/0.5A ST_2"  DQ 8x24VDC/0.5A ST
   slot 3: "DQ 8x24VDC/0.5A ST_3"  DQ 8x24VDC/0.5A ST  6ES7 132-6BF01-0BA0  V0.0
      slot 1: "DQ 8x24VDC/0.5A ST_3"  DQ 8x24VDC/0.5A ST
   slot 4: "Server module_1"  Server module  6ES7 193-6PA00-0AA0  V1.1
      slot 1: "Server module_1"  Server module
   slot 127: "BA 2xRJ45"  BA 2xRJ45  6ES7 193-6AR00-0AA0  V0.0
      slot 1: "Port_1"  6ES7 193-6AR00-0AA0  V0.0
      slot 2: "Port_2"  6ES7 193-6AR00-0AA0  V0.0
DEVICE "ET 200SP station_32"  ET 200SP-Station
   slot 0: "Rack_0"  Rack  6ES5 710-8MAx1
   slot 0: "1bx2001et200sp"  IM 155-6 PN ST  6ES7 155-6AU01-0BN0  V4.1
   slot 1: "DQ 8x24VDC/0.5A ST_1"  DQ 8x24VDC/0.5A ST  6ES7 132-6BF01-0BA0  V0.0
      slot 1: "DQ 8x24VDC/0.5A ST_1"  DQ 8x24VDC/0.5A ST
   slot 2: "DQ 8x24VDC/0.5A ST_2"  DQ 8x24VDC/0.5A ST  6ES7 132-6BF01-0BA0  V0.0
      slot 1: "DQ 8x24VDC/0.5A ST_2"  DQ 8x24VDC/0.5A ST
   slot 3: "DQ 8x24VDC/0.5A ST_3"  DQ 8x24VDC/0.5A ST  6ES7 132-6BF01-0BA0  V0.0
      slot 1: "DQ 8x24VDC/0.5A ST_3"  DQ 8x24VDC/0.5A ST
   slot 4: "Server module_1"  Server module  6ES7 193-6PA00-0AA0  V1.1
      slot 1: "Server module_1"  Server module
   slot 127: "BA 2xRJ45"  BA 2xRJ45  6ES7 193-6AR00-0AA0  V0.0
      slot 1: "Port_1"  6ES7 193-6AR00-0AA0  V0.0
      slot 2: "Port_2"  6ES7 193-6AR00-0AA0  V0.0
DEVICE "KP8_27"  SIMATIC Key Panel
   slot 0: "Rack"  Rail  V1.0
   slot 0: "1bx2001kp8"  KP8  6AV3 688-3AY36-0AX0  R01.00.00
DEVICE "ET 200SP station_33"  ET 200SP-Station
   slot 0: "Rack_0"  Rack  6ES5 710-8MAx1
   slot 0: "1bx2002et200sp"  IM 155-6 PN ST  6ES7 155-6AU01-0BN0  V4.1
   slot 1: "DQ 8x24VDC/0.5A ST_1"  DQ 8x24VDC/0.5A ST  6ES7 132-6BF01-0BA0  V0.0
      slot 1: "DQ 8x24VDC/0.5A ST_1"  DQ 8x24VDC/0.5A ST
   slot 2: "DQ 8x24VDC/0.5A ST_2"  DQ 8x24VDC/0.5A ST  6ES7 132-6BF01-0BA0  V0.0
      slot 1: "DQ 8x24VDC/0.5A ST_2"  DQ 8x24VDC/0.5A ST
   slot 3: "DQ 8x24VDC/0.5A ST_3"  DQ 8x24VDC/0.5A ST  6ES7 132-6BF01-0BA0  V0.0
      slot 1: "DQ 8x24VDC/0.5A ST_3"  DQ 8x24VDC/0.5A ST
   slot 4: "Server module_1"  Server module  6ES7 193-6PA00-0AA0  V1.1
      slot 1: "Server module_1"  Server module
   slot 127: "BA 2xRJ45"  BA 2xRJ45  6ES7 193-6AR00-0AA0  V0.0
      slot 1: "Port_1"  6ES7 193-6AR00-0AA0  V0.0
      slot 2: "Port_2"  6ES7 193-6AR00-0AA0  V0.0
DEVICE "KP8_28"  SIMATIC Key Panel
   slot 0: "Rack"  Rail  V1.0
   slot 0: "1bx2002kp8"  KP8  6AV3 688-3AY36-0AX0  R01.00.00
DEVICE "KP8_29"  SIMATIC Key Panel
   slot 0: "Rack"  Rail  V1.0
   slot 0: "1bx2003kp8"  KP8  6AV3 688-3AY36-0AX0  R01.00.00
DEVICE "ET 200SP station_34"  ET 200SP-Station
   slot 0: "Rack_0"  Rack  6ES5 710-8MAx1
   slot 0: "1bx2003et200sp"  IM 155-6 PN ST  6ES7 155-6AU01-0BN0  V4.1
   slot 1: "DQ 8x24VDC/0.5A ST_1"  DQ 8x24VDC/0.5A ST  6ES7 132-6BF01-0BA0  V0.0
      slot 1: "DQ 8x24VDC/0.5A ST_1"  DQ 8x24VDC/0.5A ST
   slot 2: "DQ 8x24VDC/0.5A ST_2"  DQ 8x24VDC/0.5A ST  6ES7 132-6BF01-0BA0  V0.0
      slot 1: "DQ 8x24VDC/0.5A ST_2"  DQ 8x24VDC/0.5A ST
   slot 3: "DQ 8x24VDC/0.5A ST_3"  DQ 8x24VDC/0.5A ST  6ES7 132-6BF01-0BA0  V0.0
      slot 1: "DQ 8x24VDC/0.5A ST_3"  DQ 8x24VDC/0.5A ST
   slot 4: "Server module_1"  Server module  6ES7 193-6PA00-0AA0  V1.1
      slot 1: "Server module_1"  Server module
   slot 127: "BA 2xRJ45"  BA 2xRJ45  6ES7 193-6AR00-0AA0  V0.0
      slot 1: "Port_1"  6ES7 193-6AR00-0AA0  V0.0
      slot 2: "Port_2"  6ES7 193-6AR00-0AA0  V0.0
DEVICE "KP8_30"  SIMATIC Key Panel
   slot 0: "Rack"  Rail  V1.0
   slot 0: "1bx2004kp8"  KP8  6AV3 688-3AY36-0AX0  R01.00.00
DEVICE "ET 200SP station_35"  ET 200SP-Station
   slot 0: "Rack_0"  Rack  6ES5 710-8MAx1
   slot 0: "1bx2004et200sp"  IM 155-6 PN ST  6ES7 155-6AU01-0BN0  V4.1
   slot 1: "DQ 8x24VDC/0.5A ST_1"  DQ 8x24VDC/0.5A ST  6ES7 132-6BF01-0BA0  V0.0
      slot 1: "DQ 8x24VDC/0.5A ST_1"  DQ 8x24VDC/0.5A ST
   slot 2: "DQ 8x24VDC/0.5A ST_2"  DQ 8x24VDC/0.5A ST  6ES7 132-6BF01-0BA0  V0.0
      slot 1: "DQ 8x24VDC/0.5A ST_2"  DQ 8x24VDC/0.5A ST
   slot 3: "DQ 8x24VDC/0.5A ST_3"  DQ 8x24VDC/0.5A ST  6ES7 132-6BF01-0BA0  V0.0
      slot 1: "DQ 8x24VDC/0.5A ST_3"  DQ 8x24VDC/0.5A ST
   slot 4: "Server module_1"  Server module  6ES7 193-6PA00-0AA0  V1.1
      slot 1: "Server module_1"  Server module
   slot 127: "BA 2xRJ45"  BA 2xRJ45  6ES7 193-6AR00-0AA0  V0.0
      slot 1: "Port_1"  6ES7 193-6AR00-0AA0  V0.0
      slot 2: "Port_2"  6ES7 193-6AR00-0AA0  V0.0
DEVICE "ET 200SP station_36"  ET 200SP-Station
   slot 0: "Rack_0"  Rack  6ES5 710-8MAx1
   slot 0: "1bx2005et200sp"  IM 155-6 PN ST  6ES7 155-6AU01-0BN0  V4.1
   slot 1: "DQ 8x24VDC/0.5A ST_1"  DQ 8x24VDC/0.5A ST  6ES7 132-6BF01-0BA0  V0.0
      slot 1: "DQ 8x24VDC/0.5A ST_1"  DQ 8x24VDC/0.5A ST
   slot 2: "DQ 8x24VDC/0.5A ST_2"  DQ 8x24VDC/0.5A ST  6ES7 132-6BF01-0BA0  V0.0
      slot 1: "DQ 8x24VDC/0.5A ST_2"  DQ 8x24VDC/0.5A ST
   slot 3: "DQ 8x24VDC/0.5A ST_3"  DQ 8x24VDC/0.5A ST  6ES7 132-6BF01-0BA0  V0.0
      slot 1: "DQ 8x24VDC/0.5A ST_3"  DQ 8x24VDC/0.5A ST
   slot 4: "Server module_1"  Server module  6ES7 193-6PA00-0AA0  V1.1
      slot 1: "Server module_1"  Server module
   slot 127: "BA 2xRJ45"  BA 2xRJ45  6ES7 193-6AR00-0AA0  V0.0
      slot 1: "Port_1"  6ES7 193-6AR00-0AA0  V0.0
      slot 2: "Port_2"  6ES7 193-6AR00-0AA0  V0.0
DEVICE "KP8_31"  SIMATIC Key Panel
   slot 0: "Rack"  Rail  V1.0
   slot 0: "1bx2005kp8"  KP8  6AV3 688-3AY36-0AX0  R01.00.00
DEVICE "KP8_32"  SIMATIC Key Panel
   slot 0: "Rack"  Rail  V1.0
   slot 0: "1bx3001kp8"  KP8  6AV3 688-3AY36-0AX0  R01.00.00
DEVICE "ET 200SP station_37"  ET 200SP-Station
   slot 0: "Rack_0"  Rack  6ES5 710-8MAx1
   slot 0: "1bx3001et200sp"  IM 155-6 PN ST  6ES7 155-6AU01-0BN0  V4.1
   slot 1: "DQ 8x24VDC/0.5A ST_1"  DQ 8x24VDC/0.5A ST  6ES7 132-6BF01-0BA0  V0.0
      slot 1: "DQ 8x24VDC/0.5A ST_1"  DQ 8x24VDC/0.5A ST
   slot 2: "DQ 8x24VDC/0.5A ST_2"  DQ 8x24VDC/0.5A ST  6ES7 132-6BF01-0BA0  V0.0
      slot 1: "DQ 8x24VDC/0.5A ST_2"  DQ 8x24VDC/0.5A ST
   slot 3: "DQ 8x24VDC/0.5A ST_3"  DQ 8x24VDC/0.5A ST  6ES7 132-6BF01-0BA0  V0.0
      slot 1: "DQ 8x24VDC/0.5A ST_3"  DQ 8x24VDC/0.5A ST
   slot 4: "Server module_1"  Server module  6ES7 193-6PA00-0AA0  V1.1
      slot 1: "Server module_1"  Server module
   slot 127: "BA 2xRJ45"  BA 2xRJ45  6ES7 193-6AR00-0AA0  V0.0
      slot 1: "Port_1"  6ES7 193-6AR00-0AA0  V0.0
      slot 2: "Port_2"  6ES7 193-6AR00-0AA0  V0.0
DEVICE "KP8_33"  SIMATIC Key Panel
   slot 0: "Rack"  Rail  V1.0
   slot 0: "1bx3002kp8"  KP8  6AV3 688-3AY36-0AX0  R01.00.00
DEVICE "ET 200SP station_38"  ET 200SP-Station
   slot 0: "Rack_0"  Rack  6ES5 710-8MAx1
   slot 0: "1bx3002et200sp"  IM 155-6 PN ST  6ES7 155-6AU01-0BN0  V4.1
   slot 1: "DQ 8x24VDC/0.5A ST_1"  DQ 8x24VDC/0.5A ST  6ES7 132-6BF01-0BA0  V0.0
      slot 1: "DQ 8x24VDC/0.5A ST_1"  DQ 8x24VDC/0.5A ST
   slot 2: "DQ 8x24VDC/0.5A ST_2"  DQ 8x24VDC/0.5A ST  6ES7 132-6BF01-0BA0  V0.0
      slot 1: "DQ 8x24VDC/0.5A ST_2"  DQ 8x24VDC/0.5A ST
   slot 3: "DQ 8x24VDC/0.5A ST_3"  DQ 8x24VDC/0.5A ST  6ES7 132-6BF01-0BA0  V0.0
      slot 1: "DQ 8x24VDC/0.5A ST_3"  DQ 8x24VDC/0.5A ST
   slot 4: "Server module_1"  Server module  6ES7 193-6PA00-0AA0  V1.1
      slot 1: "Server module_1"  Server module
   slot 127: "BA 2xRJ45"  BA 2xRJ45  6ES7 193-6AR00-0AA0  V0.0
      slot 1: "Port_1"  6ES7 193-6AR00-0AA0  V0.0
      slot 2: "Port_2"  6ES7 193-6AR00-0AA0  V0.0
DEVICE "KP8_34"  SIMATIC Key Panel
   slot 0: "Rack"  Rail  V1.0
   slot 0: "1bx3003kp8"  KP8  6AV3 688-3AY36-0AX0  R01.00.00
DEVICE "ET 200SP station_39"  ET 200SP-Station
   slot 0: "Rack_0"  Rack  6ES5 710-8MAx1
   slot 0: "1bx3003et200sp"  IM 155-6 PN ST  6ES7 155-6AU01-0BN0  V4.1
   slot 1: "DQ 8x24VDC/0.5A ST_1"  DQ 8x24VDC/0.5A ST  6ES7 132-6BF01-0BA0  V0.0
      slot 1: "DQ 8x24VDC/0.5A ST_1"  DQ 8x24VDC/0.5A ST
   slot 2: "DQ 8x24VDC/0.5A ST_2"  DQ 8x24VDC/0.5A ST  6ES7 132-6BF01-0BA0  V0.0
      slot 1: "DQ 8x24VDC/0.5A ST_2"  DQ 8x24VDC/0.5A ST
   slot 3: "DQ 8x24VDC/0.5A ST_3"  DQ 8x24VDC/0.5A ST  6ES7 132-6BF01-0BA0  V0.0
      slot 1: "DQ 8x24VDC/0.5A ST_3"  DQ 8x24VDC/0.5A ST
   slot 4: "Server module_1"  Server module  6ES7 193-6PA00-0AA0  V1.1
      slot 1: "Server module_1"  Server module
   slot 127: "BA 2xRJ45"  BA 2xRJ45  6ES7 193-6AR00-0AA0  V0.0
      slot 1: "Port_1"  6ES7 193-6AR00-0AA0  V0.0
      slot 2: "Port_2"  6ES7 193-6AR00-0AA0  V0.0
*)

// ===== PLC "PLC_1"  CPU 1517F-3 PN/DP =====

VAR_GLOBAL   // PLC tag table "Default tag table"
   "System_Byte" AT %MB1 : Byte;
   "FirstScan" AT %M1.0 : Bool;
   "DiagStatUpdt" AT %M1.1 : Bool;
   "AlwaysTRUE" AT %M1.2 : Bool;
   "AlwaysFALSE" AT %M1.3 : Bool;
   "Clock_Byte" AT %MB0 : Byte;
   "Clock_10Hz" AT %M0.0 : Bool;
   "Clock_5Hz" AT %M0.1 : Bool;
   "Clock_2.5Hz" AT %M0.2 : Bool;
   "Clock_2Hz" AT %M0.3 : Bool;
   "Clock_1.25Hz" AT %M0.4 : Bool;
   "Clock_1Hz" AT %M0.5 : Bool;
   "Clock_0.625Hz" AT %M0.6 : Bool;
   "Clock_0.5Hz" AT %M0.7 : Bool;
   "Temp Reset" AT %M2.0 : Bool;
   "clearPartData" AT %M100.0 : Bool;
   "setDefaultPresets" AT %M100.1 : Bool;
   "hardInitReq" AT %M100.2 : Bool;
   "dbg" AT %M500.0 : Bool;
   "dbgSetDefTimes" AT %M5000.0 : Bool;
END_VAR

VAR_GLOBAL CONSTANT   // PLC tag table "Default tag table"
   "1BX 2.0 01" : Int := 31;
   "1BX 2.0 02" : Int := 32;
   "1BX 2.0 03" : Int := 33;
   "1BX 2.0 04" : Int := 34;
   "1BX 2.0 05" : Int := 35;
   "1BX 3.0 01" : Int := 36;
   "1BX 3.0 02" : Int := 37;
   "1BX 3.0 03" : Int := 38;
END_VAR

VAR_GLOBAL   // PLC tag table "VOLVO 16 01"
   "VOLVO 16 01 KP8 In" AT %ID0 : DWord;
   "VOLVO 16 01 IO" AT %QD1000 : DWord;
   "VOLVO 16 01 KP8 Out" AT %QD0 : DWord;
END_VAR

VAR_GLOBAL   // PLC tag table "VOLVO 16 02"
   "VOLVO 16 02 KP8 In" AT %ID4 : DWord;
   "VOLVO 16 02 IO" AT %QD1004 : DWord;
   "VOLVO 16 02 KP8 Out" AT %QD4 : DWord;
END_VAR

VAR_GLOBAL   // PLC tag table "VOLVO 16 03"
   "VOLVO 16 03 KP8 In" AT %ID8 : DWord;
   "VOLVO 16 03 IO" AT %QD1008 : DWord;
   "VOLVO 16 03 KP8 Out" AT %QD8 : DWord;
END_VAR

VAR_GLOBAL   // PLC tag table "VOLVO 16 04"
   "VOLVO 16 04 KP8 In" AT %ID12 : DWord;
   "VOLVO 16 04 IO" AT %QD1012 : DWord;
   "VOLVO 16 04 KP8 Out" AT %QD12 : DWord;
END_VAR

VAR_GLOBAL   // PLC tag table "VOLVO 16 05"
   "VOLVO 16 05 KP8 In" AT %ID16 : DWord;
   "VOLVO 16 05 IO" AT %QD1016 : DWord;
   "VOLVO 16 05 KP8 Out" AT %QD16 : DWord;
END_VAR

VAR_GLOBAL   // PLC tag table "VOLVO 16 06"
   "VOLVO 16 06 KP8 In" AT %ID20 : DWord;
   "VOLVO 16 06 IO" AT %QD1020 : DWord;
   "VOLVO 16 06 KP8 Out" AT %QD20 : DWord;
END_VAR

VAR_GLOBAL   // PLC tag table "VOLVO 16 07"
   "VOLVO 16 07 KP8 In" AT %ID24 : DWord;
   "VOLVO 16 07 IO" AT %QD1024 : DWord;
   "VOLVO 16 07 KP8 Out" AT %QD24 : DWord;
END_VAR

VAR_GLOBAL   // PLC tag table "VOLVO 16 08"
   "VOLVO 16 08 KP8 In" AT %ID28 : DWord;
   "VOLVO 16 08 IO" AT %QD1028 : DWord;
   "VOLVO 16 08 KP8 Out" AT %QD28 : DWord;
END_VAR

VAR_GLOBAL   // PLC tag table "VOLVO 16 09"
   "VOLVO 16 09 KP8 In" AT %ID32 : DWord;
   "VOLVO 16 09 IO" AT %QD1032 : DWord;
   "VOLVO 16 09 KP8 Out" AT %QD32 : DWord;
END_VAR

VAR_GLOBAL   // PLC tag table "VOLVO 16 10"
   "VOLVO 16 10 KP8 In" AT %ID36 : DWord;
   "VOLVO 16 10 IO" AT %QD1036 : DWord;
   "VOLVO 16 10 KP8 Out" AT %QD36 : DWord;
END_VAR

VAR_GLOBAL   // PLC tag table "VOLVO 16 11"
   "VOLVO 16 11 KP8 In" AT %ID40 : DWord;
   "VOLVO 16 11 IO" AT %QD1040 : DWord;
   "VOLVO 16 11 KP8 Out" AT %QD40 : DWord;
END_VAR

VAR_GLOBAL   // PLC tag table "CHM 02"
   "CHM 02 KP8 In" AT %ID44 : DWord;
   "CHM 02 KP8 Out" AT %QD44 : DWord;
   "CHM 02 IO" AT %QD1044 : DWord;
END_VAR

VAR_GLOBAL   // PLC tag table "CHM 03"
   "CHM 03 KP8 In" AT %ID48 : DWord;
   "CHM 03 KP8 Out" AT %QD48 : DWord;
   "CHM 03 IO" AT %QD1048 : DWord;
END_VAR

VAR_GLOBAL   // PLC tag table "CHM 04"
   "CHM 04 KP8 In" AT %ID52 : DWord;
   "CHM 04 KP8 Out" AT %QD52 : DWord;
   "CHM 04 IO" AT %QD1052 : DWord;
END_VAR

VAR_GLOBAL   // PLC tag table "CHM 05"
   "CHM 05 KP8 In" AT %ID56 : DWord;
   "CHM 05 KP8 Out" AT %QD56 : DWord;
   "CHM 05 IO" AT %QD1056 : DWord;
END_VAR

VAR_GLOBAL   // PLC tag table "CDO 01"
   "CDO 01 KP8 In" AT %ID60 : DWord;
   "CDO 01 KP8 Out" AT %QD60 : DWord;
   "CDO 01 IO" AT %QD1060 : DWord;
END_VAR

VAR_GLOBAL   // PLC tag table "CDO 02"
   "CDO 02 KP8 In" AT %ID64 : DWord;
   "CDO 02 KP8 Out" AT %QD64 : DWord;
   "CDO 02 IO" AT %QD1064 : DWord;
END_VAR

VAR_GLOBAL   // PLC tag table "CDO 03"
   "CDO 03 KP8 In" AT %ID68 : DWord;
   "CDO 03 KP8 Out" AT %QD68 : DWord;
   "CDO 03 IO" AT %QD1068 : DWord;
END_VAR

VAR_GLOBAL   // PLC tag table "BFL 01"
   "BFL 01 KP8 In" AT %ID72 : DWord;
   "BFL 01 KP8 Out" AT %QD72 : DWord;
   "BFL 01 IO" AT %QD1072 : DWord;
END_VAR

VAR_GLOBAL   // PLC tag table "BFL 02"
   "BFL 02 KP8 In" AT %ID76 : DWord;
   "BFL 02 KP8 Out" AT %QD76 : DWord;
   "BFL 02 IO" AT %QD1076 : DWord;
END_VAR

VAR_GLOBAL   // PLC tag table "BFL 03"
   "BFL 03 KP8 In" AT %ID80 : DWord;
   "BFL 03 KP8 Out" AT %QD80 : DWord;
   "BFL 03 IO" AT %QD1080 : DWord;
END_VAR

VAR_GLOBAL   // PLC tag table "LGS 01"
   "LGS 01 KP8 In" AT %ID84 : DWord;
   "LGS 01 KP8 Out" AT %QD84 : DWord;
   "LGS 01 IO" AT %QD1084 : DWord;
END_VAR

VAR_GLOBAL   // PLC tag table "LGS 02"
   "LGS 02 KP8 In" AT %ID88 : DWord;
   "LGS 02 KP8 Out" AT %QD88 : DWord;
   "LGS 02 IO" AT %QD1088 : DWord;
END_VAR

VAR_GLOBAL   // PLC tag table "CHM 01"
   "CHM 01 KP8 In" AT %ID92 : DWord;
   "CHM 01 IO" AT %QD1092 : DWord;
   "CHM 01 KP8 Out" AT %QD92 : DWord;
END_VAR

VAR_GLOBAL CONSTANT   // PLC tag table "Color Library"
   "BkBk" : USInt := 0;
   "BgWh" : USInt := 1;
   "FgWh" : USInt := 2;
   "FlWh" : USInt := 3;
   "BgGray" : USInt := 4;
   "FgGray" : USInt := 5;
   "FlGray" : USInt := 6;
   "BgLRd" : USInt := 7;
   "FgLRd" : USInt := 8;
   "FlLRd" : USInt := 9;
   "BgDRd" : USInt := 10;
   "FgDRd" : USInt := 11;
   "FlDrd" : USInt := 12;
   "BgLYe" : USInt := 13;
   "FgLYe" : USInt := 14;
   "FlLYe" : USInt := 15;
   "BgDYe" : USInt := 16;
   "FgDYe" : USInt := 17;
   "FlDYe" : USInt := 18;
   "BgLGr" : USInt := 19;
   "FgLGr" : USInt := 20;
   "FlLGr" : USInt := 21;
   "BgDGr" : USInt := 22;
   "FgDGr" : USInt := 23;
   "FlDGr" : USInt := 24;
   "BgLTe" : USInt := 25;
   "FgLTe" : USInt := 26;
   "FlLTe" : USInt := 27;
   "BgDTe" : USInt := 28;
   "FgDTe" : USInt := 29;
   "FlDTe" : USInt := 30;
   "BgLBl" : USInt := 31;
   "FgLBl" : USInt := 32;
   "FlLBl" : USInt := 33;
   "BgDBl" : USInt := 34;
   "FgDBl" : USInt := 35;
   "FlDBl" : USInt := 36;
   "BgLPu" : USInt := 37;
   "FgLPu" : USInt := 38;   // foreground light purple
   "FlLPu" : USInt := 39;
   "BgDPu" : USInt := 40;
   "FgDPu" : USInt := 41;
   "FlDPu" : USInt := 42;
   "disabled" : USInt := 254;
   "invisible" : USInt := 255;
   "LBlDRd" : USInt := 43;
   "DRdLBl" : USInt := 44;
   "LBlDRdFl" : USInt := 45;
   "DBlDRd" : USInt := 46;
   "DRdDBl" : USInt := 47;
   "DBlDRdFl" : USInt := 48;
END_VAR

VAR_GLOBAL CONSTANT   // PLC tag table "Comm Diag"
   "pnioDeviceCount" : Int := 48;   // Upper limit of devices per HMI screen
   "USERDIAG_SLOTS_PER_SCREEN_UPPER_LIM" : Int := 31;   // Upper limit of slots per HMI screen
   "USERDIAG_SLOTS_PER_DEVICE_UPPER_LIM" : Int := 31;   // max number of modules per device
   "USERDIAG_DEVICES_PER_IO_SYSTEM_UPPER_LIM" : Int := 128;   // Upper limit of devices/slaves per IO-System/DP-Mastersystem
   "USERDIAG_SLOTS_PER_PLC_UPPER_LIM" : Int := 31;   // max number of local modules
   "USERDIAG_IO_SYSTEMS_UPPER_LIM" : Int := 1;   // Upper limit of IO-Systems/DP-Mastersystems
   "USERDIAG_IOSYSTEM_1" : Int := 1;   // Index for first IO-System/DP-Mastersystem
END_VAR

VAR_GLOBAL   // PLC tag table "Simulation"
   "simMode" AT %M100.3 : Bool;
END_VAR

VAR_GLOBAL CONSTANT   // PLC tag table "Simulation"
   "simKP8Count" : Int := 11;
END_VAR

VAR_GLOBAL CONSTANT   // PLC tag table "Station Meta Data"
   "ptsPerStn" : Int := 7;
   "stnCount" : Int := 38;
   "defaultAlotted" : Real := 1800.0;
   "defaultCritical" : Real := 300.0;
   "menuCntPerStn" : Int := 49;
   "mStringLen" : Int := 40;
   "sStringLen" : Int := 20;
   "lStringLen" : Int := 60;
END_VAR

VAR_GLOBAL CONSTANT   // PLC tag table "Station IDs"
   "VOLVO 16 01" : Int := 0;
   "VOLVO 16 02" : Int := 1;
   "VOLVO 16 03" : Int := 2;
   "VOLVO 16 04" : Int := 3;
   "VOLVO 16 05" : Int := 4;
   "VOLVO 16 06" : Int := 5;
   "VOLVO 16 07" : Int := 6;
   "VOLVO 16 08" : Int := 7;
   "VOLVO 16 09" : Int := 8;
   "VOLVO 16 10" : Int := 9;
   "VOLVO 16 11" : Int := 10;
   "CHM 01" : Int := 11;
   "CHM 02" : Int := 12;
   "CHM 03" : Int := 13;
   "CHM 04" : Int := 14;
   "CHM 05" : Int := 15;
   "CDO 01" : Int := 16;
   "CDO 02" : Int := 17;
   "CDO 03" : Int := 18;
   "BFL 01" : Int := 19;
   "BFL 02" : Int := 20;
   "BFL 03" : Int := 21;
   "LGS 01" : Int := 22;
   "LGS 02" : Int := 23;
   "LGS 03" : Int := 24;
   "CV 01" : Int := 25;
   "CV 02" : Int := 26;
   "CV 03" : Int := 27;
   "CV 04" : Int := 28;
   "PC 01" : Int := 29;
   "PC 02" : Int := 30;
END_VAR

VAR_GLOBAL CONSTANT   // PLC tag table "HMI Part Request Screen"
   "partReqHmiRowCount" : Int := 11;   // number of rows displayed on hmi
END_VAR

VAR_GLOBAL CONSTANT   // PLC tag table "HMI Settings Screen"
   "hmiSelStnCount" : Int := 11;   // labels for settings screen
END_VAR

VAR_GLOBAL CONSTANT   // PLC tag table "Part Request Data Base"
   "partReqDataRowCount" : Int := 199;
END_VAR

VAR_GLOBAL CONSTANT   // PLC tag table "LED Sign"
   "ledRowCount" : Int := 11;
END_VAR

VAR_GLOBAL CONSTANT   // PLC tag table "HMI Select Station"
   "hmiStnCount" : Int := 4;   // number of stations using basic panel instead of kp8 (-1 for array)
   "hmiStnPartSelScrnBtnCnt" : Int := 7;   // number of buttons on part select screen (-1 for array)
   "hmiStnMenuSelScrnBtnCnt" : Int := 29;   // number of buttons on menu select screen (short and long rows use different data, -1 for array)
   "hmiStnMenuSelLblCnt" : Int := 29;   // number of labels (2 per row, short & long rows use same data, - 1 for array)
   "hmiStnTmpltBtnCnt" : Int := 1;   // number of button on the template (-1 for array)
END_VAR

VAR_GLOBAL   // PLC tag table "LGS 03"
   "LGS 03 KP8 In" AT %ID96 : DWord;
   "LGS 03 IO" AT %QD1096 : DWord;
   "LGS 03 KP8 Out" AT %QD96 : DWord;
END_VAR

VAR_GLOBAL   // PLC tag table "CV 01"
   "CV 01 KP8 In" AT %ID100 : DWord;
   "CV 01 IO" AT %QD1100 : DWord;
   "CV 01 KP8 Out" AT %QD100 : DWord;
END_VAR

VAR_GLOBAL   // PLC tag table "CV 02"
   "CV 02 KP8 In" AT %ID104 : DWord;
   "CV 02 IO" AT %QD1104 : DWord;
   "CV 02 KP8 Out" AT %QD104 : DWord;
END_VAR

VAR_GLOBAL   // PLC tag table "CV 03"
   "CV 03 KP8 In" AT %ID108 : DWord;
   "CV 03 IO" AT %QD1108 : DWord;
   "CV 03 KP8 Out" AT %QD108 : DWord;
END_VAR

VAR_GLOBAL   // PLC tag table "CV 04"
   "CV 04 KP8 In" AT %ID112 : DWord;
   "CV 04 IO" AT %QD1112 : DWord;
   "CV 04 KP8 Out" AT %QD112 : DWord;
END_VAR

VAR_GLOBAL   // PLC tag table "PC 01"
   "PC 01 KP8 In" AT %ID116 : DWord;
   "PC 01 IO" AT %QD1116 : DWord;
   "PC 01 KP8 Out" AT %QD116 : DWord;
END_VAR

VAR_GLOBAL   // PLC tag table "PC 02"
   "PC 02 KP8 In" AT %ID120 : DWord;
   "PC 02 IO" AT %QD1120 : DWord;
   "PC 02 KP8 Out" AT %QD120 : DWord;
END_VAR

VAR_GLOBAL   // PLC tag table "1BX 2.0 01"
   "1BX 2.0 01 KP8 In" AT %ID124 : DWord;
   "1BX 2.0 01 KP8 Out" AT %QD124 : DWord;
   "1BX 2.0 01 IO" AT %QD1124 : DWord;
END_VAR

VAR_GLOBAL   // PLC tag table "1BX 2.0 02"
   "1BX 2.0 02 KP8 In" AT %ID128 : DWord;
   "1BX 2.0 02 KP8 Out" AT %QD128 : DWord;
   "1BX 2.0 02 IO" AT %QD1128 : DWord;
END_VAR

VAR_GLOBAL   // PLC tag table "1BX 2.0 03"
   "1BX 2.0 03 KP8 In" AT %ID132 : DWord;
   "1BX 2.0 03 KP8 Out" AT %QD132 : DWord;
   "1BX 2.0 03 IO" AT %QD1132 : DWord;
END_VAR

VAR_GLOBAL   // PLC tag table "1BX 2.0 04"
   "1BX 2.0 04 KP8 In" AT %ID136 : DWord;
   "1BX 2.0 04 KP8 Out" AT %QD136 : DWord;
   "1BX 2.0 04 IO" AT %QD1136 : DWord;
END_VAR

VAR_GLOBAL   // PLC tag table "1BX 2.0 05"
   "1BX 2.0 05 KP8 In" AT %ID140 : DWord;
   "1BX 2.0 05 KP8 Out" AT %QD140 : DWord;
   "1BX 2.0 05 IO" AT %QD1140 : DWord;
END_VAR

VAR_GLOBAL   // PLC tag table "1BX 3.0 01"
   "1BX 3.0 01 KP8 In" AT %ID144 : DWord;
   "1BX 3.0 01 KP8 Out" AT %QD144 : DWord;
   "1BX 3.0 01 IO" AT %QD1144 : DWord;
END_VAR

VAR_GLOBAL   // PLC tag table "1BX 3.0 02"
   "1BX 3.0 02 KP8 In" AT %ID148 : DWord;
   "1BX 3.0 02 KP8 Out" AT %QD148 : DWord;
   "1BX 3.0 02 IO" AT %QD1148 : DWord;
END_VAR

VAR_GLOBAL   // PLC tag table "1BX 3.0 03"
   "1BX 3.0 03 KP8 In" AT %ID152 : DWord;
   "1BX 3.0 03 KP8 Out" AT %QD152 : DWord;
   "1BX 3.0 03 IO" AT %QD1152 : DWord;
END_VAR

TYPE "Stations"
VERSION : 0.1
   STRUCT
      me : Array[0.."stnCount"] of "Station";
   END_STRUCT;
END_TYPE

TYPE "Part Call Screen"
VERSION : 0.1
   STRUCT
      row : Array[0.."partReqHmiRowCount"] of "Table Row";
   END_STRUCT;
END_TYPE

TYPE "Part Req Log Row"
VERSION : 0.1
   STRUCT
      address : Int;
      reqType : Int;
      timeStamp : DTL;
   END_STRUCT;
END_TYPE

TYPE "Barcode Screen"
VERSION : 0.1
   STRUCT
      partNumber : WString[40];
      barcode : String;
      orderCancelled : Bool;
      ordered : Bool;
   END_STRUCT;
END_TYPE

TYPE "Table Row"
VERSION : 0.1
   STRUCT
      address : UInt;
      ordered : Bool;
      pbSelection : Struct
         actuate : Bool;
         animate : USInt;
      END_STRUCT;
      rtBackground : Struct
         animate : USInt;
      END_STRUCT;
      tfDropZone : Struct
         animate : USInt;
         value : WString[20];
      END_STRUCT;
      tfLine : Struct
         animate : USInt;
         value : WString[20];
      END_STRUCT;
      tfPartNumber : Struct
         animateDL : USInt;
         animateSL : USInt;
         value : WString[40];
      END_STRUCT;
      tfTime : Struct
         animate : USInt;
         value : WString[20];
      END_STRUCT;
   END_STRUCT;
END_TYPE

TYPE "Runtime Data"
VERSION : 0.1
   STRUCT
      asReal : Real;
      elapsed : LReal;
      mem : LReal;
   END_STRUCT;
END_TYPE

TYPE "KP8 Button Config"
VERSION : 0.1
   STRUCT
      activate : Array[0.."ptsPerStn"] of Bool;
      colorOn1 : Array[0.."ptsPerStn"] of String[10];
      colorOn2 : Array[0.."ptsPerStn"] of String[10];
      colorOff : Array[0.."ptsPerStn"] of String[10];
      flash : Array[0.."ptsPerStn"] of Bool;
      group : Array[0.."ptsPerStn"] of Int;
      mode : Array[0.."ptsPerStn"] of Bool;
   END_STRUCT;
END_TYPE

TYPE "Elapsed Time"
VERSION : 0.1
   STRUCT
      partReq : Array[0.."ptsPerStn"] of Real;
      resetReq : Real;
   END_STRUCT;
END_TYPE

TYPE "Part Request Data"
VERSION : 0.1
   STRUCT
      row : Array[0.."partReqDataRowCount"] of "Table Row";
   END_STRUCT;
END_TYPE

TYPE "Station"
VERSION : 0.1
   STRUCT
      animations : Array[0.."ptsPerStn"] of Int;
      btnStates : Array[0.."ptsPerStn"] of Bool;
      dropZone : USInt;
      elapsedTime : "Elapsed Time";
      groupSelect : Int;
      kp8Config : "KP8 Button Config";
      kp8In : Byte;
      kp8Out : DWord;
      init : "Station Initialization";
      line : WString[20];
      partNumbers : Array[0.."ptsPerStn"] of WString["mStringLen"];
      partOrdered : Array[0.."ptsPerStn"] of Bool;
      partRequested : Array[0.."ptsPerStn"] of Bool;
      presetTime : "Preset Time";
      settings : "Station Settings Screen";
      stackLightOut : DWord;
   END_STRUCT;
END_TYPE

TYPE "Settings"
VERSION : 0.1
   STRUCT
      alotted : Struct
         assign : "PB Data: Text Label";
         ioField : "IO Field Data: Timers";
      END_STRUCT;
      critical : Struct
         assign : "PB Data: Text Label";
         ioField : "IO Field Data: Timers";
      END_STRUCT;
      kp8 : Struct
         selectButtons : "PB Data: Text Label";
         btnSelState : Array[0.."ptsPerStn"] of Bool;
         buttons : Array[0.."ptsPerStn"] of "PB Data: Text Label";
         selBtnNumber : Int;
         selCount : Int;
      END_STRUCT;
      stations : Struct
         selectAll : "PB Data: Text Label";
         nextGroup : "PB Data: Graphic/Text List";
         prevGroup : "PB Data: Graphic/Text List";
         selectBtns : Array[0.."hmiSelStnCount"] of "PB Data: Text Label";
         selCount : Int;
         selNumber : Int;
      END_STRUCT;
      partNumber : Struct
         assign : "PB Data: Text Label";
         ioField : "IO Field Data: Part Number";
      END_STRUCT;
      viewingStation : Struct
         btns : Array[0.."ptsPerStn"] of "Station Assignment: Button Details";
         dzData : "Drop Zone Data";
         lineData : "Line Label Data";
         next : "PB Data: Graphic/Text List";
         previous : "PB Data: Graphic/Text List";
         "name" : WString[20];
      END_STRUCT;
   END_STRUCT;
END_TYPE

TYPE "PB Data: Graphic/Text List"
VERSION : 0.1
   STRUCT
      actuate : Bool;
      animate : USInt;
      listSelect : UInt;
   END_STRUCT;
END_TYPE

TYPE "LED Sign Data"
VERSION : 0.1
   STRUCT
      row : Array[0.."ledRowCount"] of "Table Row";
   END_STRUCT;
END_TYPE

TYPE "PB Data: Text Label"
VERSION : 0.1
   STRUCT
      actuate : Bool;
      animate : USInt;
      label : WString[20];
   END_STRUCT;
END_TYPE

TYPE "Station Old Presses"
VERSION : 0.1
   STRUCT
      me : Array[0.."stnCount", 0.."ptsPerStn"] of Bool;
   END_STRUCT;
END_TYPE

TYPE "Station Assignment: Button Details"
VERSION : 0.1
   STRUCT
      alloted : Struct
         animate : USInt;
         value : WString[10];
      END_STRUCT;
      critical : Struct
         animate : USInt;
         value : WString[10];
      END_STRUCT;
      label : Struct
         animate : USInt;
         value : WString[2];
      END_STRUCT;
      partNumber : Struct
         animate : USInt;
         value : WString[40];
      END_STRUCT;
      select : Struct
         actuate : Bool;
         animate : USInt;
      END_STRUCT;
   END_STRUCT;
END_TYPE

TYPE "IO Field Data: Part Number"
VERSION : 0.1
   STRUCT
      animate : USInt;
      inputFinished : Bool;
      value : WString[40];
   END_STRUCT;
END_TYPE

TYPE "Line Label Data"
VERSION : 0.1
   STRUCT
      animate : Struct
         bg : USInt;
         ioField : USInt;
      END_STRUCT;
      inputFinished : Bool;
      value : WString[10];
   END_STRUCT;
END_TYPE

TYPE "Drop Zone Data"
VERSION : 0.1
   STRUCT
      animate : Struct
         bg : USInt;
         ioField : USInt;
      END_STRUCT;
      inputFinished : Bool;
      value : WString[10];
   END_STRUCT;
END_TYPE

TYPE "IO Field Data: Timers"
VERSION : 0.1
   STRUCT
      animate : USInt;
      inputFinished : Bool;
      value : WString[5];
   END_STRUCT;
END_TYPE

TYPE "Table Nav"
VERSION : 0.1
   STRUCT
      top : "PB Data: Graphic/Text List";
      pageUp : "PB Data: Graphic/Text List";
      lineUp : "PB Data: Graphic/Text List";
      lineDown : "PB Data: Graphic/Text List";
      pageDown : "PB Data: Graphic/Text List";
      bottom : "PB Data: Graphic/Text List";
   END_STRUCT;
END_TYPE

TYPE "Station Sim Data"
VERSION : 0.1
   STRUCT
      stn : Struct
         animate : USInt;
         label : WString[20];
      END_STRUCT;
      btn : Struct
         actuate : Byte;
         animate : Array[0..7] of USInt;
         labels : Array[0..7] of WString [4];
      END_STRUCT;
   END_STRUCT;
END_TYPE

TYPE "Simulated Stations"
VERSION : 0.1
   STRUCT
      down : "PB Data: Graphic/Text List";
      firstStn : Int;
      me : Array[0.."simKP8Count"] of "Station Sim Data";
      up : "PB Data: Graphic/Text List";
   END_STRUCT;
END_TYPE

TYPE "Part Req Log"
VERSION : 0.1
   STRUCT
      me : Array[0..99] of "Part Req Log Row";
   END_STRUCT;
END_TYPE

TYPE "HSS: Part Selection Screen"
VERSION : 0.1
   STRUCT
      animate : Array[0.."hmiStnPartSelScrnBtnCnt"] of Int;
      pbs : DWord;
      txt : Array[0.."hmiStnPartSelScrnBtnCnt"] of WString [40];
   END_STRUCT;
END_TYPE

TYPE "UserDiag_typeSlot"
VERSION : 0.1
   STRUCT
      hardwareId : Hw_Io := 16#0000;   // Hardware identifier of the module which is inserted in the slot
      state : USInt := 0;   // Status of the device/slave. 1:ok; 2:faulty, 3:lost connection, 4:disabled, 5:problem, 12:was faulty, 13:was lost, 14:was disabled, 15:problem gone
      exists : Bool := FALSE;   // TRUE: Modul is existing
      configured : Bool := FALSE;   // TRUE: Modul is configured
      faulty : Bool := FALSE;   // TRUE: Modul is faulty
      problem : Bool := FALSE;   // TRUE: Modul has a problem
      disabled : Bool := FALSE;   // TRUE: Modul is disabled
      error : Bool := FALSE;   // TRUE: Error in module which is inserted in the slot
   END_STRUCT;
END_TYPE

TYPE "UserDiag_typePLC"
VERSION : 0.1
   STRUCT
      hardwareId : Hw_Device := 16#0000;   // Hardware identifier of the PLC
      error : Bool := FALSE;   // TRUE: Error in PLC
      actualConfiguredSlots : Int := 0;   // Number of configured local slots at PLC
      slots : Array[0.."USERDIAG_SLOTS_PER_PLC_UPPER_LIM"] of "UserDiag_typeSlot";   // Information of the PLC slots; index = slotnumber; PLC always at slot 1
   END_STRUCT;
END_TYPE

TYPE "UserDiag_typeDevice"
VERSION : 0.1
   STRUCT
      hardwareId : Hw_Device := 16#0000;   // Hardware identifier of the device/slave
      number : UInt := 0;   // Profinet device number/Profibus address of the slave
      "name" : WString[20] := WSTRING#'';   // Name of the device/slave
      ipAddress : IP_V4;   // IP address of the device
      state : USInt := 0;   // Status of the device/slave. 1:ok; 2:faulty, 3:lost connection, 4:disabled, 5:problem, 12:was faulty, 13:was lost, 14:was disabled, 15:problem gone
      exists : Bool := FALSE;   // TRUE: Device/slave is existing
      configured : Bool := FALSE;   // TRUE: Device/slave is configured
      faulty : Bool := FALSE;   // TRUE: Device/slave is faulty
      problem : Bool := FALSE;   // TRUE: Device/slave has a problem
      disabled : Bool := FALSE;   // TRUE: Device/slave is disabled
      error : Bool := FALSE;   // TRUE: Error in device/slave
      nextDevice : Int := 0;   // device number of next device
      actualConfiguredSlots : Int := 0;   // Number of configured slots in the device/slave
      slots : Array[0.."USERDIAG_SLOTS_PER_DEVICE_UPPER_LIM"] of "UserDiag_typeSlot";   // Slot information of a device/slave
   END_STRUCT;
END_TYPE

TYPE "UserDiag_typeIOSystem"
VERSION : 0.1
   STRUCT
      hardwareId : Hw_IoSystem := 16#0000;   // Hardware identifier of the IO-System/DP-Mastersystem
      number : UInt := 0;   // IO-System/DP-Mastersystem number
      error : Bool := FALSE;   // TRUE: Error in IO-System/DP-Mastersystem
      firstDevice : Int := 0;   // device number (index) of first device in IO System
      lastDevice : Int := 0;   // device number (index) of last device IO System
      actualConfiguredDevices : Int := 0;   // Number of configured devices/slaves in IO-System/DP-Mastersystem
      devices : Array[1.."USERDIAG_DEVICES_PER_IO_SYSTEM_UPPER_LIM"] of "UserDiag_typeDevice";   // Device/Slave information
   END_STRUCT;
END_TYPE

TYPE "Network Health Screen"
VERSION : 0.1
   STRUCT
      et200spPopUp : "Station: ET200SP Comm Debug Data";
      kp8PopUp : "Station: KP8 Comm Debug Data";
      pnioDevices : Array[1.."pnioDeviceCount"] of "PB Data: Text Label";
      selectedDevice : Int;
   END_STRUCT;
   // // pnioDevices[1] : volvo1601kp8
   // // pnioDevices[2] : volvo1601et200sp
   // // pnioDevices[3] : volvo1602kp8
   // // pnioDevices[4] : volvo1602et200sp
   // // pnioDevices[5] : volvo1603kp8
   // // pnioDevices[6] : volvo1603et200sp
   // // pnioDevices[7] : volvo1604kp8
   // // pnioDevices[8] : volvo1604et200sp
   // // pnioDevices[9] : volvo1605kp8
   // // pnioDevices[10] : volvo1605et200sp
   // // pnioDevices[11] : volvo1606kp8
   // // pnioDevices[12] : volvo1606et200sp
   // // pnioDevices[13] : volvo1607kp8
   // // pnioDevices[14] : volvo1607et200sp
   // // pnioDevices[15] : volvo1608kp8
   // // pnioDevices[16] : volvo1608et200sp
   // // pnioDevices[17] : volvo1609kp8
   // // pnioDevices[18] : volvo1609et200sp
   // // pnioDevices[19] : volvo1610kp8
   // // pnioDevices[20] : volvo1610et200sp
   // // pnioDevices[21] : volvo1611kp8
   // // pnioDevices[22] : volvo1611et200sp
   // // pnioDevices[23] : chm01kp8
   // // pnioDevices[24] : chm01et200sp
   // // pnioDevices[25] : chm02kp8
   // // pnioDevices[26] : chm02et200sp
   // // pnioDevices[27] : chm03kp8
   // // pnioDevices[28] : chm03et200sp
   // // pnioDevices[29] : chm04kp8
   // // pnioDevices[30] : chm04et200sp
   // // pnioDevices[31] : chm05kp8
   // // pnioDevices[32] : chm05et200sp
   // // pnioDevices[33] : cd001kp8
   // // pnioDevices[34] : cd001et200sp
   // // pnioDevices[35] : cd002kp8
   // // pnioDevices[36] : cd002et200sp
   // // pnioDevices[37] : cd003kp8
   // // pnioDevices[38] : cd003et200sp
   // // pnioDevices[39] : bfl01kp8
   // // pnioDevices[40] : bfl01et200sp
   // // pnioDevices[41] : bfl02kp8
   // // pnioDevices[42] : bfl02et200sp
   // // pnioDevices[43] : bfl03kp8
   // // pnioDevices[44] : bfl03et200sp
   // // pnioDevices[45] : lgs01kp8
   // // pnioDevices[46] : lgs01et200sp
   // // pnioDevices[47] : lgs02kp8
   // // pnioDevices[48] : lgs02et200sp
END_TYPE

TYPE "UserDiag_typeActIOSystem"
VERSION : 0.1
   STRUCT
      actIOSystemNumber : Int := 1;   // Number of actual selected IO-system/DP-Mastersystem
      actIODeviceNumbers : Array[1.."pnioDeviceCount"] of UInt;   // Device numbers/profibus addresses of actual selected IO-System/DP-Mastersystem
      actIODeviceState : Array[1.."pnioDeviceCount"] of USInt;   // State of devices/slaves in actual selected IO-System/DP-Mastersystem
      actDeviceSlotsUsed : Array[0.."USERDIAG_SLOTS_PER_SCREEN_UPPER_LIM"] of Bool;   // Used slots of actual selected device/slave
      actDeviceSlotsState : Array[0.."USERDIAG_SLOTS_PER_SCREEN_UPPER_LIM"] of USInt;   // States of actual selected device/slave
   END_STRUCT;
END_TYPE

TYPE "Station: ET200SP Comm Debug Data"
VERSION : 0.1
   STRUCT
      dismissPB : Bool;
      IM : "ET200SP: IM Data";
      DQ01 : "ET200SP: DQ Data";
      DQ02 : "ET200SP: DQ Data";
      DQ03 : "ET200SP: DQ Data";
      profinetName : Struct
         animate : USInt;
         label : WString[20];
      END_STRUCT;
      serverModule : "ET200SP: Server Module Data";
   END_STRUCT;
END_TYPE

TYPE "ET200SP: IM Data"
VERSION : 0.1
   STRUCT
      bg : USInt;
      error : USInt;
      lnk01 : USInt;
      lnk02 : USInt;
      maint : USInt;
      pwr : USInt;
      run : USInt;
   END_STRUCT;
END_TYPE

TYPE "ET200SP: DQ Data"
VERSION : 0.1
   STRUCT
      bg : USInt;
      bgTem : USInt;
      diag : USInt;
      pwr : USInt;
      x0 : USInt;
      x1 : USInt;
      x2 : USInt;
      x3 : USInt;
      x4 : USInt;
      x5 : USInt;
      x6 : USInt;
      x7 : USInt;
   END_STRUCT;
END_TYPE

TYPE "ET200SP: Server Module Data"
VERSION : 0.1
   STRUCT
      bg : USInt;
   END_STRUCT;
END_TYPE

TYPE "Station: KP8 Comm Debug Data"
VERSION : 0.1
   STRUCT
      dismissPB : Bool;
      profinetName : Struct
         animate : USInt;
         label : WString[20];
      END_STRUCT;
      stencilBackground : USInt;
      X1P1 : Struct
         transmit : USInt;
         receive : USInt;
      END_STRUCT;
      X1P2 : Struct
         transmit : USInt;
         receive : USInt;
      END_STRUCT;
   END_STRUCT;
END_TYPE

TYPE "Recipe: Libraries"
VERSION : 0.1
   STRUCT
      stations : Array[0.."stnCount"] of "Recipe: Library";
   END_STRUCT;
END_TYPE

TYPE "Station Initialization"
VERSION : 0.1
   STRUCT
      hard : Bool;
      soft : Bool;
   END_STRUCT;
END_TYPE

TYPE "Preset Time"
VERSION : 0.1
   STRUCT
      allotted : Array[0.."ptsPerStn"] of Real;
      critical : Array[0.."ptsPerStn"] of Real;
   END_STRUCT;
END_TYPE

TYPE "Station Settings Screen"
VERSION : 0.1
   STRUCT
      selected : Bool;
      btnSelection : Array[0.."ptsPerStn"] of Bool;
   END_STRUCT;
END_TYPE

TYPE "HSS: Compressed"
VERSION : 0.1
   STRUCT
      scrnSlctPrt : "HSS: Part Selection Screen";
      scrnSlctMn : "HSS: Menu Selection Screen";
      scrnTmplt : "HSS: Template Screen";
   END_STRUCT;
END_TYPE

TYPE "HSS: Menu Selection Screen"
VERSION : 0.1
   STRUCT
      animate : Array[0.."hmiStnMenuSelScrnBtnCnt"] of Int;
      pbs : DWord;
      txt : Array[0.."hmiStnMenuSelLblCnt"] of WString ["lStringLen"];
   END_STRUCT;
END_TYPE

TYPE "HSS: Template Screen"
VERSION : 0.1
   STRUCT
      animate : Array[0.."hmiStnTmpltBtnCnt"] of Int;
      pb : DWord;
      text : Array[0.."hmiStnTmpltBtnCnt"] of WString ["lStringLen"];
   END_STRUCT;
END_TYPE

TYPE "Recipe: Library"
VERSION : 0.1
   STRUCT
      size : Int;
      wip : Array[0.."menuCntPerStn"] of WString["lStringLen"];
      raw : Array[0.."menuCntPerStn", 0.."ptsPerStn"] of WString["mStringLen"];
   END_STRUCT;
END_TYPE

